LIN {X 0,Y 198.707,Z 605.472,A -85,B 0,C 180,E1 -21893.443,E2 -21893.443} C_VEL
LIN {X 0,Y 202.396,Z 597.043,A -85,B 0,C 180,E1 -21896.831,E2 -21896.831} C_VEL
LIN {X 0,Y 206.089,Z 588.246,A -85,B 0,C 180,E1 -21899.631,E2 -21899.631} C_VEL
LIN {X 0,Y 209.473,Z 579.533,A -85,B 0,C 180,E1 -21901.895,E2 -21901.895} C_VEL
LIN {X 0,Y 213.628,Z 567.883,A -85,B 0,C 180,E1 -21904.308,E2 -21904.308} C_VEL
LIN {X 0,Y 217.053,Z 556.425,A -85,B 0,C 180,E1 -21906.218,E2 -21906.218} C_VEL
LIN {X 0,Y 220.359,Z 543.729,A -85,B 0,C 180,E1 -21907.872,E2 -21907.872} C_VEL
LIN {X 0,Y 223.315,Z 530.569,A -85,B 0,C 180,E1 -21909.149,E2 -21909.149} C_VEL
LIN {X 0,Y 225.4,Z 517.843,A -85,B 0,C 180,E1 -21910.091,E2 -21910.091} C_VEL
LIN {X 0,Y 227.124,Z 503.349,A -85,B 0,C 180,E1 -21910.82,E2 -21910.82} C_VEL
LIN {X 0,Y 231.055,Z 437.728,A -85,B 0,C 180,E1 -21912.715,E2 -21912.715} C_VEL
LIN {X 0,Y 231.07,Z 434.373,A -85,B 0,C 180,E1 -21912.851,E2 -21912.851} C_VEL
LIN {X 0,Y 224.582,Z 419.408,A -85,B 0,C 180,E1 -21915.069,E2 -21915.069} C_VEL
LIN {X 0,Y 218.217,Z 406.943,A -85,B 0,C 180,E1 -21917.363,E2 -21917.363} C_VEL
LIN {X 0,Y 214.281,Z 400.305,A -85,B 0,C 180,E1 -21918.851,E2 -21918.851} C_VEL
LIN {X 0,Y 209.411,Z 393.182,A -85,B 0,C 180,E1 -21920.78,E2 -21920.78} C_VEL
LIN {X 0,Y 206.167,Z 388.687,A -85,B 0,C 180,E1 -21922.149,E2 -21922.149} C_VEL
LIN {X 0,Y 203.479,Z 384.928,A -85,B 0,C 180,E1 -21923.353,E2 -21923.353} C_VEL
LIN {X 0,Y 200.868,Z 381.448,A -85,B 0,C 180,E1 -21924.578,E2 -21924.578} C_VEL
LIN {X 0,Y 199.915,Z 380.302,A -85,B 0,C 180,E1 -21925.035,E2 -21925.035} C_VEL
LIN {X 0,Y 197.517,Z 377.514,A -85,B 0,C 180,E1 -21926.222,E2 -21926.222} C_VEL
LIN {X 0,Y 196.503,Z 375.589,A -85,B 0,C 180,E1 -21926.793,E2 -21926.793} C_VEL
LIN {X 0,Y 194.099,Z 373.615,A -85,B 0,C 180,E1 -21928.031,E2 -21928.031} C_VEL
LIN {X 0,Y 192.852,Z 371.337,A -85,B 0,C 180,E1 -21928.79,E2 -21928.79} C_VEL
LIN {X 0,Y 192.566,Z 370.108,A -85,B 0,C 180,E1 -21929.044,E2 -21929.044} C_VEL
LIN {X 0,Y 192.61,Z 370.098,A -85,B 0,C 180,E1 -21931.683,E2 -21931.683} C_VEL
LIN {X 0,Y 192.662,Z 370.106,A -85,B 0,C 180,E1 -21936.343,E2 -21936.343} C_VEL
LIN {X 0,Y 192.683,Z 370.072,A -85,B 0,C 180,E1 -21941.49,E2 -21941.49} C_VEL
LIN {X 0,Y 192.723,Z 370.103,A -85,B 0,C 180,E1 -21945.21,E2 -21945.21} C_VEL
LIN {X 0,Y 192.933,Z 370.075,A -85,B 0,C 180,E1 -21949.566,E2 -21949.566} C_VEL
LIN {X 0,Y 192.953,Z 370.074,A -85,B 0,C 180,E1 -21953.727,E2 -21953.727} C_VEL
LIN {X 0,Y 193.218,Z 370.043,A -85,B 0,C 180,E1 -21957.915,E2 -21957.915} C_VEL
LIN {X 0,Y 193.4,Z 370.008,A -85,B 0,C 180,E1 -21960,E2 -21960} C_VEL
LIN {X 0,Y 192.923,Z 370.068,A -85,B 0,C 180,E1 -21964.178,E2 -21964.178} C_VEL
LIN {X 0,Y 193.011,Z 370.058,A -85,B 0,C 180,E1 -21968.375,E2 -21968.375} C_VEL
LIN {X 0,Y 192.778,Z 370.087,A -85,B 0,C 180,E1 -21972.635,E2 -21972.635} C_VEL
LIN {X 0,Y 192.704,Z 370.097,A -85,B 0,C 180,E1 -21976.963,E2 -21976.963} C_VEL
LIN {X 0,Y 192.561,Z 370.092,A -85,B 0,C 180,E1 -21981.406,E2 -21981.406} C_VEL
LIN {X 0,Y 192.599,Z 370.097,A -85,B 0,C 180,E1 -21984.19,E2 -21984.19} C_VEL
LIN {X 0,Y 192.589,Z 370.093,A -85,B 0,C 180,E1 -21988.866,E2 -21988.866} C_VEL
LIN {X 0,Y 192.562,Z 370.11,A -85,B 0,C 180,E1 -21990.88,E2 -21990.88} C_VEL
LIN {X 0,Y 193.417,Z 372.657,A -85,B 0,C 180,E1 -21991.489,E2 -21991.489} C_VEL
LIN {X 0,Y 193.705,Z 373.112,A -85,B 0,C 180,E1 -21991.659,E2 -21991.659} C_VEL
LIN {X 0,Y 196.21,Z 378.545,A -85,B 0,C 180,E1 -21993.181,E2 -21993.181} C_VEL
LIN {X 0,Y 202.441,Z 393.008,A -85,B 0,C 180,E1 -21996.634,E2 -21996.634} C_VEL
LIN {X 0,Y 203.994,Z 395.569,A -85,B 0,C 180,E1 -21997.361,E2 -21997.361} C_VEL
LIN {X 0,Y 210.292,Z 406.349,A -85,B 0,C 180,E1 -22000.114,E2 -22000.114} C_VEL
LIN {X 0,Y 216.539,Z 418.079,A -85,B 0,C 180,E1 -22002.6,E2 -22002.6} C_VEL
LIN {X 0,Y 222.539,Z 431.217,A -85,B 0,C 180,E1 -22004.843,E2 -22004.843} C_VEL
LIN {X 0,Y 225.822,Z 439.404,A -85,B 0,C 180,E1 -22006.029,E2 -22006.029} C_VEL
LIN {X 0,Y 221.988,Z 502.379,A -85,B 0,C 180,E1 -22007.846,E2 -22007.846} C_VEL
LIN {X 0,Y 220.45,Z 517.246,A -85,B 0,C 180,E1 -22008.513,E2 -22008.513} C_VEL
LIN {X 0,Y 218.354,Z 529.758,A -85,B 0,C 180,E1 -22009.329,E2 -22009.329} C_VEL
LIN {X 0,Y 215.954,Z 540.985,A -85,B 0,C 180,E1 -22010.311,E2 -22010.311} C_VEL
LIN {X 0,Y 212.766,Z 553.433,A -85,B 0,C 180,E1 -22011.736,E2 -22011.736} C_VEL
LIN {X 0,Y 209.227,Z 565.16,A -85,B 0,C 180,E1 -22013.464,E2 -22013.464} C_VEL
LIN {X 0,Y 205.398,Z 576.632,A -85,B 0,C 180,E1 -22015.632,E2 -22015.632} C_VEL
LIN {X 0,Y 201.599,Z 586.349,A -85,B 0,C 180,E1 -22017.888,E2 -22017.888} C_VEL
LIN {X 0,Y 197.502,Z 596.069,A -85,B 0,C 180,E1 -22020.71,E2 -22020.71} C_VEL
LIN {X 0,Y 193.869,Z 604.134,A -85,B 0,C 180,E1 -22023.639,E2 -22023.639} C_VEL
LIN {X 0,Y 190.425,Z 611.727,A -85,B 0,C 180,E1 -22027.125,E2 -22027.125} C_VEL
LIN {X 0,Y 188.014,Z 617.259,A -85,B 0,C 180,E1 -22030.345,E2 -22030.345} C_VEL
LIN {X 0,Y 185.449,Z 622.939,A -85,B 0,C 180,E1 -22034.62,E2 -22034.62} C_VEL
LIN {X 0,Y 183.947,Z 627.063,A -85,B 0,C 180,E1 -22038.99,E2 -22038.99} C_VEL
LIN {X 0,Y 183.189,Z 629.751,A -85,B 0,C 180,E1 -22043.394,E2 -22043.394} C_VEL
LIN {X 0,Y 182.991,Z 631.077,A -85,B 0,C 180,E1 -22047.802,E2 -22047.802} C_VEL
LIN {X 0,Y 183.062,Z 631.239,A -85,B 0,C 180,E1 -22050.003,E2 -22050.003} C_VEL
LIN {X 0,Y 183.019,Z 630.557,A -85,B 0,C 180,E1 -22054.408,E2 -22054.408} C_VEL
LIN {X 0,Y 183.498,Z 628.531,A -85,B 0,C 180,E1 -22058.816,E2 -22058.816} C_VEL
LIN {X 0,Y 184.614,Z 625.117,A -85,B 0,C 180,E1 -22063.207,E2 -22063.207} C_VEL
LIN {X 0,Y 186.675,Z 620.215,A -85,B 0,C 180,E1 -22067.532,E2 -22067.532} C_VEL
LIN {X 0,Y 189.593,Z 613.67,A -85,B 0,C 180,E1 -22071.761,E2 -22071.761} C_VEL
LIN {X 0,Y 193.917,Z 611.789,A -85,B 0,C 180,E1 -22075.783,E2 -22075.783} C_VEL
LIN {X 0,Y 199.616,Z 608.772,A -85,B 0,C 180,E1 -22079.535,E2 -22079.535} C_VEL
LIN {X 0,Y 206.41,Z 604.439,A -85,B 0,C 180,E1 -22083.013,E2 -22083.013} C_VEL
LIN {X 0,Y 214.305,Z 598.674,A -85,B 0,C 180,E1 -22086.181,E2 -22086.181} C_VEL
LIN {X 0,Y 223.09,Z 591.287,A -85,B 0,C 180,E1 -22089.058,E2 -22089.058} C_VEL
LIN {X 0,Y 232.751,Z 582.111,A -85,B 0,C 180,E1 -22091.631,E2 -22091.631} C_VEL
LIN {X 0,Y 241.882,Z 572.221,A -85,B 0,C 180,E1 -22093.638,E2 -22093.638} C_VEL
LIN {X 0,Y 250.221,Z 562.013,A -85,B 0,C 180,E1 -22095.165,E2 -22095.165} C_VEL
LIN {X 0,Y 257.281,Z 552.141,A -85,B 0,C 180,E1 -22096.279,E2 -22096.279} C_VEL
LIN {X 0,Y 257.573,Z 551.734,A -85,B 0,C 180,E1 -22096.657,E2 -22096.657} C_VEL
LIN {X 0,Y 250.018,Z 562.221,A -85,B 0,C 180,E1 -22098.117,E2 -22098.117} C_VEL
LIN {X 0,Y 242.233,Z 571.531,A -85,B 0,C 180,E1 -22099.793,E2 -22099.793} C_VEL
LIN {X 0,Y 233.601,Z 580.397,A -85,B 0,C 180,E1 -22101.921,E2 -22101.921} C_VEL
LIN {X 0,Y 225.099,Z 587.859,A -85,B 0,C 180,E1 -22104.335,E2 -22104.335} C_VEL
LIN {X 0,Y 217.934,Z 593.201,A -85,B 0,C 180,E1 -22106.755,E2 -22106.755} C_VEL
LIN {X 0,Y 210.044,Z 598.033,A -85,B 0,C 180,E1 -22109.875,E2 -22109.875} C_VEL
LIN {X 0,Y 203.096,Z 601.298,A -85,B 0,C 180,E1 -22113.266,E2 -22113.266} C_VEL
LIN {X 0,Y 197.064,Z 603.056,A -85,B 0,C 180,E1 -22116.903,E2 -22116.903} C_VEL
LIN {X 0,Y 192.029,Z 603.407,A -85,B 0,C 180,E1 -22120.769,E2 -22120.769} C_VEL
LIN {X 0,Y 188.438,Z 602.296,A -85,B 0,C 180,E1 -22124.866,E2 -22124.866} C_VEL
LIN {X 0,Y 185.775,Z 599.724,A -85,B 0,C 180,E1 -22129.097,E2 -22129.097} C_VEL
LIN {X 0,Y 184.203,Z 595.669,A -85,B 0,C 180,E1 -22133.428,E2 -22133.428} C_VEL
LIN {X 0,Y 183.814,Z 591.518,A -85,B 0,C 180,E1 -22136.712,E2 -22136.712} C_VEL
LIN {X 0,Y 183.676,Z 585.283,A -85,B 0,C 180,E1 -22140.548,E2 -22140.548} C_VEL
LIN {X 0,Y 183.852,Z 578.541,A -85,B 0,C 180,E1 -22143.836,E2 -22143.836} C_VEL
LIN {X 0,Y 184.278,Z 570.082,A -85,B 0,C 180,E1 -22147.175,E2 -22147.175} C_VEL
LIN {X 0,Y 184.92,Z 559.88,A -85,B 0,C 180,E1 -22150.401,E2 -22150.401} C_VEL
LIN {X 0,Y 185.69,Z 549.274,A -85,B 0,C 180,E1 -22153.126,E2 -22153.126} C_VEL
LIN {X 0,Y 186.702,Z 537.558,A -85,B 0,C 180,E1 -22155.558,E2 -22155.558} C_VEL
LIN {X 0,Y 187.729,Z 524.558,A -85,B 0,C 180,E1 -22157.709,E2 -22157.709} C_VEL
LIN {X 0,Y 188.701,Z 510.981,A -85,B 0,C 180,E1 -22159.443,E2 -22159.443} C_VEL
LIN {X 0,Y 189.583,Z 495.968,A -85,B 0,C 180,E1 -22160.833,E2 -22160.833} C_VEL
LIN {X 0,Y 193.383,Z 417.044,A -85,B 0,C 180,E1 -22166.116,E2 -22166.116} C_VEL
LIN {X 0,Y 191.04,Z 396.091,A -85,B 0,C 180,E1 -22167.576,E2 -22167.576} C_VEL
LIN {X 0,Y 188.706,Z 385.709,A -85,B 0,C 180,E1 -22168.414,E2 -22168.414} C_VEL
LIN {X 0,Y 187.873,Z 381.706,A -85,B 0,C 180,E1 -22169.657,E2 -22169.657} C_VEL
LIN {X 0,Y 188.604,Z 383.232,A -85,B 0,C 180,E1 -22170.16,E2 -22170.16} C_VEL
LIN {X 0,Y 189.272,Z 383.585,A -85,B 0,C 180,E1 -22170.533,E2 -22170.533} C_VEL
LIN {X 0,Y 191.035,Z 383.228,A -85,B 0,C 180,E1 -22171.395,E2 -22171.395} C_VEL
LIN {X 0,Y 192.098,Z 382.434,A -85,B 0,C 180,E1 -22171.858,E2 -22171.858} C_VEL
LIN {X 0,Y 194.344,Z 382.672,A -85,B 0,C 180,E1 -22172.927,E2 -22172.927} C_VEL
LIN {X 0,Y 197.017,Z 386.201,A -85,B 0,C 180,E1 -22174.338,E2 -22174.338} C_VEL
LIN {X 0,Y 198.275,Z 387.839,A -85,B 0,C 180,E1 -22174.97,E2 -22174.97} C_VEL
LIN {X 0,Y 201.836,Z 392.677,A -85,B 0,C 180,E1 -22176.678,E2 -22176.678} C_VEL
LIN {X 0,Y 207.332,Z 400.427,A -85,B 0,C 180,E1 -22179.097,E2 -22179.097} C_VEL
LIN {X 0,Y 212.843,Z 409.078,A -85,B 0,C 180,E1 -22181.33,E2 -22181.33} C_VEL
LIN {X 0,Y 219.414,Z 422.009,A -85,B 0,C 180,E1 -22183.854,E2 -22183.854} C_VEL
LIN {X 0,Y 224.284,Z 433.17,A -85,B 0,C 180,E1 -22185.63,E2 -22185.63} C_VEL
LIN {X 0,Y 225.739,Z 436.684,A -85,B 0,C 180,E1 -22186.144,E2 -22186.144} C_VEL
LIN {X 0,Y 223.107,Z 481.871,A -85,B 0,C 180,E1 -22187.457,E2 -22187.457} C_VEL
LIN {X 0,Y 221.59,Z 504.39,A -85,B 0,C 180,E1 -22188.162,E2 -22188.162} C_VEL
LIN {X 0,Y 219.962,Z 517.73,A -85,B 0,C 180,E1 -22188.85,E2 -22188.85} C_VEL
LIN {X 0,Y 217.444,Z 531.634,A -85,B 0,C 180,E1 -22189.876,E2 -22189.876} C_VEL
LIN {X 0,Y 214.505,Z 544.565,A -85,B 0,C 180,E1 -22191.197,E2 -22191.197} C_VEL
LIN {X 0,Y 211.033,Z 557.109,A -85,B 0,C 180,E1 -22192.868,E2 -22192.868} C_VEL
LIN {X 0,Y 207.451,Z 568.548,A -85,B 0,C 180,E1 -22194.833,E2 -22194.833} C_VEL
LIN {X 0,Y 203.572,Z 579.047,A -85,B 0,C 180,E1 -22197.058,E2 -22197.058} C_VEL
LIN {X 0,Y 200.001,Z 587.851,A -85,B 0,C 180,E1 -22199.365,E2 -22199.365} C_VEL
LIN {X 0,Y 196.155,Z 596.725,A -85,B 0,C 180,E1 -22202.237,E2 -22202.237} C_VEL
LIN {X 0,Y 192.286,Z 605.219,A -85,B 0,C 180,E1 -22205.718,E2 -22205.718} C_VEL
LIN {X 0,Y 189.301,Z 612.061,A -85,B 0,C 180,E1 -22209.344,E2 -22209.344} C_VEL
LIN {X 0,Y 187.046,Z 616.782,A -85,B 0,C 180,E1 -22212.504,E2 -22212.504} C_VEL
LIN {X 0,Y 184.936,Z 621.666,A -85,B 0,C 180,E1 -22216.817,E2 -22216.817} C_VEL
LIN {X 0,Y 183.702,Z 625.064,A -85,B 0,C 180,E1 -22221.194,E2 -22221.194} C_VEL
LIN {X 0,Y 183.125,Z 627.082,A -85,B 0,C 180,E1 -22225.595,E2 -22225.595} C_VEL
LIN {X 0,Y 183.07,Z 627.769,A -85,B 0,C 180,E1 -22229.997,E2 -22229.997} C_VEL
LIN {X 0,Y 183.123,Z 627.138,A -85,B 0,C 180,E1 -22234.399,E2 -22234.399} C_VEL
LIN {X 0,Y 183.681,Z 625.172,A -85,B 0,C 180,E1 -22238.8,E2 -22238.8} C_VEL
LIN {X 0,Y 184.896,Z 621.821,A -85,B 0,C 180,E1 -22243.18,E2 -22243.18} C_VEL
LIN {X 0,Y 187.015,Z 616.983,A -85,B 0,C 180,E1 -22247.492,E2 -22247.492} C_VEL
LIN {X 0,Y 189.191,Z 612.318,A -85,B 0,C 180,E1 -22250.661,E2 -22250.661} C_VEL
LIN {X 0,Y 192.191,Z 605.537,A -85,B 0,C 180,E1 -22254.288,E2 -22254.288} C_VEL
LIN {X 0,Y 196.076,Z 597.108,A -85,B 0,C 180,E1 -22257.769,E2 -22257.769} C_VEL
LIN {X 0,Y 199.924,Z 588.311,A -85,B 0,C 180,E1 -22260.641,E2 -22260.641} C_VEL
LIN {X 0,Y 203.474,Z 579.598,A -85,B 0,C 180,E1 -22262.953,E2 -22262.953} C_VEL
LIN {X 0,Y 207.381,Z 569.207,A -85,B 0,C 180,E1 -22265.174,E2 -22265.174} C_VEL
LIN {X 0,Y 210.943,Z 557.912,A -85,B 0,C 180,E1 -22267.143,E2 -22267.143} C_VEL
LIN {X 0,Y 214.35,Z 545.556,A -85,B 0,C 180,E1 -22268.829,E2 -22268.829} C_VEL
LIN {X 0,Y 217.371,Z 532.887,A -85,B 0,C 180,E1 -22270.133,E2 -22270.133} C_VEL
LIN {X 0,Y 219.793,Z 519.423,A -85,B 0,C 180,E1 -22271.181,E2 -22271.181} C_VEL
LIN {X 0,Y 221.572,Z 505.563,A -85,B 0,C 180,E1 -22271.927,E2 -22271.927} C_VEL
LIN {X 0,Y 223.066,Z 485.36,A -85,B 0,C 180,E1 -22272.567,E2 -22272.567} C_VEL
LIN {X 0,Y 225.873,Z 436.775,A -85,B 0,C 180,E1 -22273.984,E2 -22273.984} C_VEL
LIN {X 0,Y 219.558,Z 422.15,A -85,B 0,C 180,E1 -22276.274,E2 -22276.274} C_VEL
LIN {X 0,Y 212.497,Z 408.401,A -85,B 0,C 180,E1 -22278.995,E2 -22278.995} C_VEL
LIN {X 0,Y 206.716,Z 399.463,A -85,B 0,C 180,E1 -22281.362,E2 -22281.362} C_VEL
LIN {X 0,Y 200.489,Z 390.766,A -85,B 0,C 180,E1 -22284.168,E2 -22284.168} C_VEL
LIN {X 0,Y 197.112,Z 386.299,A -85,B 0,C 180,E1 -22285.836,E2 -22285.836} C_VEL
LIN {X 0,Y 194.47,Z 382.927,A -85,B 0,C 180,E1 -22287.227,E2 -22287.227} C_VEL
LIN {X 0,Y 193.636,Z 381.69,A -85,B 0,C 180,E1 -22287.697,E2 -22287.697} C_VEL
LIN {X 0,Y 191.036,Z 378.928,A -85,B 0,C 180,E1 -22289.153,E2 -22289.153} C_VEL
LIN {X 0,Y 189.725,Z 376.624,A -85,B 0,C 180,E1 -22289.994,E2 -22289.994} C_VEL
LIN {X 0,Y 187.341,Z 374.834,A -85,B 0,C 180,E1 -22291.425,E2 -22291.425} C_VEL
LIN {X 0,Y 185.853,Z 372.39,A -85,B 0,C 180,E1 -22292.48,E2 -22292.48} C_VEL
LIN {X 0,Y 185.509,Z 370.971,A -85,B 0,C 180,E1 -22292.883,E2 -22292.883} C_VEL
LIN {X 0,Y 185.57,Z 370.973,A -85,B 0,C 180,E1 -22295.38,E2 -22295.38} C_VEL
LIN {X 0,Y 185.614,Z 370.95,A -85,B 0,C 180,E1 -22301.177,E2 -22301.177} C_VEL
LIN {X 0,Y 185.652,Z 370.986,A -85,B 0,C 180,E1 -22304.633,E2 -22304.633} C_VEL
LIN {X 0,Y 185.876,Z 370.955,A -85,B 0,C 180,E1 -22309.418,E2 -22309.418} C_VEL
LIN {X 0,Y 185.918,Z 370.952,A -85,B 0,C 180,E1 -22313.488,E2 -22313.488} C_VEL
LIN {X 0,Y 186.164,Z 370.922,A -85,B 0,C 180,E1 -22317.836,E2 -22317.836} C_VEL
LIN {X 0,Y 186.366,Z 370.884,A -85,B 0,C 180,E1 -22320,E2 -22320} C_VEL
LIN {X 0,Y 185.871,Z 370.946,A -85,B 0,C 180,E1 -22324.337,E2 -22324.337} C_VEL
LIN {X 0,Y 185.961,Z 370.936,A -85,B 0,C 180,E1 -22328.695,E2 -22328.695} C_VEL
LIN {X 0,Y 185.704,Z 370.968,A -85,B 0,C 180,E1 -22333.125,E2 -22333.125} C_VEL
LIN {X 0,Y 185.641,Z 370.978,A -85,B 0,C 180,E1 -22337.63,E2 -22337.63} C_VEL
LIN {X 0,Y 185.528,Z 370.965,A -85,B 0,C 180,E1 -22342.26,E2 -22342.26} C_VEL
LIN {X 0,Y 185.513,Z 371.02,A -85,B 0,C 180,E1 -22347.116,E2 -22347.116} C_VEL
LIN {X 0,Y 186.269,Z 373.389,A -85,B 0,C 180,E1 -22347.758,E2 -22347.758} C_VEL
LIN {X 0,Y 188.414,Z 375.851,A -85,B 0,C 180,E1 -22349.159,E2 -22349.159} C_VEL
LIN {X 0,Y 189.937,Z 376.846,A -85,B 0,C 180,E1 -22350.045,E2 -22350.045} C_VEL
LIN {X 0,Y 191.839,Z 380.019,A -85,B 0,C 180,E1 -22351.236,E2 -22351.236} C_VEL
LIN {X 0,Y 194.171,Z 382.365,A -85,B 0,C 180,E1 -22352.509,E2 -22352.509} C_VEL
LIN {X 0,Y 196.68,Z 385.884,A -85,B 0,C 180,E1 -22353.863,E2 -22353.863} C_VEL
LIN {X 0,Y 198.116,Z 387.577,A -85,B 0,C 180,E1 -22354.582,E2 -22354.582} C_VEL
LIN {X 0,Y 201.825,Z 392.601,A -85,B 0,C 180,E1 -22356.375,E2 -22356.375} C_VEL
LIN {X 0,Y 203.994,Z 395.569,A -85,B 0,C 180,E1 -22357.361,E2 -22357.361} C_VEL
LIN {X 0,Y 206.102,Z 399.752,A -85,B 0,C 180,E1 -22358.352,E2 -22358.352} C_VEL
LIN {X 0,Y 207.66,Z 404.671,A -85,B 0,C 180,E1 -22359.155,E2 -22359.155} C_VEL
LIN {X 0,Y 211.072,Z 418.814,A -85,B 0,C 180,E1 -22361.001,E2 -22361.001} C_VEL
LIN {X 0,Y 212.243,Z 422.12,A -85,B 0,C 180,E1 -22361.528,E2 -22361.528} C_VEL
LIN {X 0,Y 217.855,Z 434.676,A -85,B 0,C 180,E1 -22363.755,E2 -22363.755} C_VEL
LIN {X 0,Y 220.59,Z 441.582,A -85,B 0,C 180,E1 -22364.803,E2 -22364.803} C_VEL
LIN {X 0,Y 217.065,Z 498.535,A -85,B 0,C 180,E1 -22366.462,E2 -22366.462} C_VEL
LIN {X 0,Y 215.781,Z 512.612,A -85,B 0,C 180,E1 -22367.009,E2 -22367.009} C_VEL
LIN {X 0,Y 213.471,Z 527.097,A -85,B 0,C 180,E1 -22367.876,E2 -22367.876} C_VEL
LIN {X 0,Y 210.538,Z 540.924,A -85,B 0,C 180,E1 -22369.077,E2 -22369.077} C_VEL
LIN {X 0,Y 207.238,Z 553.371,A -85,B 0,C 180,E1 -22370.52,E2 -22370.52} C_VEL
LIN {X 0,Y 203.199,Z 566.134,A -85,B 0,C 180,E1 -22372.445,E2 -22372.445} C_VEL
LIN {X 0,Y 199.14,Z 577.725,A -85,B 0,C 180,E1 -22374.726,E2 -22374.726} C_VEL
LIN {X 0,Y 194.825,Z 588.067,A -85,B 0,C 180,E1 -22377.245,E2 -22377.245} C_VEL
LIN {X 0,Y 190.651,Z 597.489,A -85,B 0,C 180,E1 -22380.159,E2 -22380.159} C_VEL
LIN {X 0,Y 186.357,Z 606.463,A -85,B 0,C 180,E1 -22383.701,E2 -22383.701} C_VEL
LIN {X 0,Y 182.895,Z 613.717,A -85,B 0,C 180,E1 -22387.406,E2 -22387.406} C_VEL
LIN {X 0,Y 180.578,Z 618.802,A -85,B 0,C 180,E1 -22390.686,E2 -22390.686} C_VEL
LIN {X 0,Y 178.065,Z 624.051,A -85,B 0,C 180,E1 -22395.138,E2 -22395.138} C_VEL
LIN {X 0,Y 176.951,Z 626.996,A -85,B 0,C 180,E1 -22398.549,E2 -22398.549} C_VEL
LIN {X 0,Y 176.121,Z 629.684,A -85,B 0,C 180,E1 -22403.128,E2 -22403.128} C_VEL
LIN {X 0,Y 175.886,Z 631.01,A -85,B 0,C 180,E1 -22407.713,E2 -22407.713} C_VEL
LIN {X 0,Y 175.974,Z 631.172,A -85,B 0,C 180,E1 -22410.003,E2 -22410.003} C_VEL
LIN {X 0,Y 175.942,Z 630.489,A -85,B 0,C 180,E1 -22414.586,E2 -22414.586} C_VEL
LIN {X 0,Y 176.456,Z 628.463,A -85,B 0,C 180,E1 -22419.17,E2 -22419.17} C_VEL
LIN {X 0,Y 177.669,Z 625.049,A -85,B 0,C 180,E1 -22423.733,E2 -22423.733} C_VEL
LIN {X 0,Y 179.889,Z 620.147,A -85,B 0,C 180,E1 -22428.216,E2 -22428.216} C_VEL
LIN {X 0,Y 182.95,Z 613.6,A -85,B 0,C 180,E1 -22432.594,E2 -22432.594} C_VEL
LIN {X 0,Y 183.345,Z 613.131,A -85,B 0,C 180,E1 -22433.078,E2 -22433.078} C_VEL
LIN {X 0,Y 187.556,Z 611.935,A -85,B 0,C 180,E1 -22436.725,E2 -22436.725} C_VEL
LIN {X 0,Y 193.492,Z 609.399,A -85,B 0,C 180,E1 -22440.568,E2 -22440.568} C_VEL
LIN {X 0,Y 200.573,Z 605.603,A -85,B 0,C 180,E1 -22444.103,E2 -22444.103} C_VEL
LIN {X 0,Y 208.767,Z 600.448,A -85,B 0,C 180,E1 -22447.301,E2 -22447.301} C_VEL
LIN {X 0,Y 217.872,Z 593.752,A -85,B 0,C 180,E1 -22450.18,E2 -22450.18} C_VEL
LIN {X 0,Y 227.814,Z 585.408,A -85,B 0,C 180,E1 -22452.745,E2 -22452.745} C_VEL
LIN {X 0,Y 236.067,Z 577.561,A -85,B 0,C 180,E1 -22454.519,E2 -22454.519} C_VEL
LIN {X 0,Y 245.567,Z 567.308,A -85,B 0,C 180,E1 -22456.232,E2 -22456.232} C_VEL
LIN {X 0,Y 246.939,Z 565.744,A -85,B 0,C 180,E1 -22456.447,E2 -22456.447} C_VEL
LIN {X 0,Y 246.766,Z 565.945,A -85,B 0,C 180,E1 -22456.88,E2 -22456.88} C_VEL
LIN {X 0,Y 237.376,Z 575.964,A -85,B 0,C 180,E1 -22458.795,E2 -22458.795} C_VEL
LIN {X 0,Y 228.45,Z 584.03,A -85,B 0,C 180,E1 -22460.901,E2 -22460.901} C_VEL
LIN {X 0,Y 219.702,Z 590.763,A -85,B 0,C 180,E1 -22463.318,E2 -22463.318} C_VEL
LIN {X 0,Y 212.302,Z 595.566,A -85,B 0,C 180,E1 -22465.753,E2 -22465.753} C_VEL
LIN {X 0,Y 204.104,Z 599.804,A -85,B 0,C 180,E1 -22468.902,E2 -22468.902} C_VEL
LIN {X 0,Y 196.881,Z 602.546,A -85,B 0,C 180,E1 -22472.351,E2 -22472.351} C_VEL
LIN {X 0,Y 190.595,Z 603.849,A -85,B 0,C 180,E1 -22476.07,E2 -22476.07} C_VEL
LIN {X 0,Y 185.351,Z 603.725,A -85,B 0,C 180,E1 -22480.047,E2 -22480.047} C_VEL
LIN {X 0,Y 181.613,Z 602.206,A -85,B 0,C 180,E1 -22484.283,E2 -22484.283} C_VEL
LIN {X 0,Y 178.844,Z 599.248,A -85,B 0,C 180,E1 -22488.669,E2 -22488.669} C_VEL
LIN {X 0,Y 177.224,Z 594.76,A -85,B 0,C 180,E1 -22493.168,E2 -22493.168} C_VEL
LIN {X 0,Y 176.834,Z 590.321,A -85,B 0,C 180,E1 -22496.582,E2 -22496.582} C_VEL
LIN {X 0,Y 176.706,Z 583.717,A -85,B 0,C 180,E1 -22500.57,E2 -22500.57} C_VEL
LIN {X 0,Y 176.888,Z 576.582,A -85,B 0,C 180,E1 -22503.987,E2 -22503.987} C_VEL
LIN {X 0,Y 177.34,Z 567.678,A -85,B 0,C 180,E1 -22507.43,E2 -22507.43} C_VEL
LIN {X 0,Y 177.931,Z 558.851,A -85,B 0,C 180,E1 -22510.239,E2 -22510.239} C_VEL
LIN {X 0,Y 178.726,Z 547.953,A -85,B 0,C 180,E1 -22513.068,E2 -22513.068} C_VEL
LIN {X 0,Y 179.734,Z 536.008,A -85,B 0,C 180,E1 -22515.595,E2 -22515.595} C_VEL
LIN {X 0,Y 180.8,Z 522.531,A -85,B 0,C 180,E1 -22517.825,E2 -22517.825} C_VEL
LIN {X 0,Y 181.786,Z 508.23,A -85,B 0,C 180,E1 -22519.625,E2 -22519.625} C_VEL
LIN {X 0,Y 182.545,Z 494.845,A -85,B 0,C 180,E1 -22520.863,E2 -22520.863} C_VEL
LIN {X 0,Y 186.308,Z 417.588,A -85,B 0,C 180,E1 -22526.292,E2 -22526.292} C_VEL
LIN {X 0,Y 184.132,Z 397.564,A -85,B 0,C 180,E1 -22527.74,E2 -22527.74} C_VEL
LIN {X 0,Y 183.291,Z 393.818,A -85,B 0,C 180,E1 -22528.033,E2 -22528.033} C_VEL
LIN {X 0,Y 183.836,Z 394.891,A -85,B 0,C 180,E1 -22528.438,E2 -22528.438} C_VEL
LIN {X 0,Y 185.317,Z 394.673,A -85,B 0,C 180,E1 -22529.258,E2 -22529.258} C_VEL
LIN {X 0,Y 186.79,Z 392.34,A -85,B 0,C 180,E1 -22529.882,E2 -22529.882} C_VEL
LIN {X 0,Y 187.698,Z 390.454,A -85,B 0,C 180,E1 -22530.222,E2 -22530.222} C_VEL
LIN {X 0,Y 190.479,Z 390.401,A -85,B 0,C 180,E1 -22531.63,E2 -22531.63} C_VEL
LIN {X 0,Y 192.248,Z 389.61,A -85,B 0,C 180,E1 -22532.424,E2 -22532.424} C_VEL
LIN {X 0,Y 195.629,Z 394.039,A -85,B 0,C 180,E1 -22534.241,E2 -22534.241} C_VEL
LIN {X 0,Y 199.148,Z 398.873,A -85,B 0,C 180,E1 -22535.999,E2 -22535.999} C_VEL
LIN {X 0,Y 206.019,Z 408.894,A -85,B 0,C 180,E1 -22539.106,E2 -22539.106} C_VEL
LIN {X 0,Y 210.05,Z 415.918,A -85,B 0,C 180,E1 -22540.806,E2 -22540.806} C_VEL
LIN {X 0,Y 216.135,Z 428.322,A -85,B 0,C 180,E1 -22543.24,E2 -22543.24} C_VEL
LIN {X 0,Y 220.586,Z 439.117,A -85,B 0,C 180,E1 -22544.949,E2 -22544.949} C_VEL
LIN {X 0,Y 216.585,Z 502.522,A -85,B 0,C 180,E1 -22546.832,E2 -22546.832} C_VEL
LIN {X 0,Y 214.902,Z 516.282,A -85,B 0,C 180,E1 -22547.502,E2 -22547.502} C_VEL
LIN {X 0,Y 212.298,Z 530.58,A -85,B 0,C 180,E1 -22548.537,E2 -22548.537} C_VEL
LIN {X 0,Y 209.478,Z 542.875,A -85,B 0,C 180,E1 -22549.768,E2 -22549.768} C_VEL
LIN {X 0,Y 205.826,Z 555.757,A -85,B 0,C 180,E1 -22551.45,E2 -22551.45} C_VEL
LIN {X 0,Y 202.387,Z 566.646,A -85,B 0,C 180,E1 -22553.296,E2 -22553.296} C_VEL
LIN {X 0,Y 198.44,Z 577.17,A -85,B 0,C 180,E1 -22555.479,E2 -22555.479} C_VEL
LIN {X 0,Y 194.579,Z 586.298,A -85,B 0,C 180,E1 -22557.805,E2 -22557.805} C_VEL
LIN {X 0,Y 190.539,Z 595.443,A -85,B 0,C 180,E1 -22560.74,E2 -22560.74} C_VEL
LIN {X 0,Y 186.885,Z 603.062,A -85,B 0,C 180,E1 -22563.773,E2 -22563.773} C_VEL
LIN {X 0,Y 183.481,Z 610.326,A -85,B 0,C 180,E1 -22567.475,E2 -22567.475} C_VEL
LIN {X 0,Y 181.021,Z 615.412,A -85,B 0,C 180,E1 -22570.728,E2 -22570.728} C_VEL
LIN {X 0,Y 178.958,Z 619.488,A -85,B 0,C 180,E1 -22574.041,E2 -22574.041} C_VEL
LIN {X 0,Y 177.234,Z 623.611,A -85,B 0,C 180,E1 -22578.561,E2 -22578.561} C_VEL
LIN {X 0,Y 176.319,Z 626.308,A -85,B 0,C 180,E1 -22583.129,E2 -22583.129} C_VEL
LIN {X 0,Y 175.95,Z 627.658,A -85,B 0,C 180,E1 -22587.707,E2 -22587.707} C_VEL
LIN {X 0,Y 175.983,Z 627.836,A -85,B 0,C 180,E1 -22589.997,E2 -22589.997} C_VEL
LIN {X 0,Y 176.034,Z 627.205,A -85,B 0,C 180,E1 -22594.576,E2 -22594.576} C_VEL
LIN {X 0,Y 176.313,Z 626.391,A -85,B 0,C 180,E1 -22596.864,E2 -22596.864} C_VEL
LIN {X 0,Y 177.205,Z 623.742,A -85,B 0,C 180,E1 -22601.434,E2 -22601.434} C_VEL
LIN {X 0,Y 178.927,Z 619.663,A -85,B 0,C 180,E1 -22605.955,E2 -22605.955} C_VEL
LIN {X 0,Y 181.755,Z 614.03,A -85,B 0,C 180,E1 -22610.362,E2 -22610.362} C_VEL
LIN {X 0,Y 184.417,Z 608.237,A -85,B 0,C 180,E1 -22613.847,E2 -22613.847} C_VEL
LIN {X 0,Y 187.949,Z 600.999,A -85,B 0,C 180,E1 -22617.258,E2 -22617.258} C_VEL
LIN {X 0,Y 191.751,Z 592.98,A -85,B 0,C 180,E1 -22620.258,E2 -22620.258} C_VEL
LIN {X 0,Y 196.031,Z 583.309,A -85,B 0,C 180,E1 -22623.139,E2 -22623.139} C_VEL
LIN {X 0,Y 200.381,Z 572.573,A -85,B 0,C 180,E1 -22625.664,E2 -22625.664} C_VEL
LIN {X 0,Y 204.13,Z 561.583,A -85,B 0,C 180,E1 -22627.759,E2 -22627.759} C_VEL
LIN {X 0,Y 207.98,Z 548.982,A -85,B 0,C 180,E1 -22629.625,E2 -22629.625} C_VEL
LIN {X 0,Y 211.223,Z 536.203,A -85,B 0,C 180,E1 -22631.078,E2 -22631.078} C_VEL
LIN {X 0,Y 213.886,Z 523.163,A -85,B 0,C 180,E1 -22632.182,E2 -22632.182} C_VEL
LIN {X 0,Y 215.997,Z 509.188,A -85,B 0,C 180,E1 -22633.017,E2 -22633.017} C_VEL
LIN {X 0,Y 217.292,Z 494.603,A -85,B 0,C 180,E1 -22633.569,E2 -22633.569} C_VEL
LIN {X 0,Y 220.743,Z 439.206,A -85,B 0,C 180,E1 -22635.176,E2 -22635.176} C_VEL
LIN {X 0,Y 215.121,Z 426.013,A -85,B 0,C 180,E1 -22637.339,E2 -22637.339} C_VEL
LIN {X 0,Y 208.292,Z 412.541,A -85,B 0,C 180,E1 -22640.127,E2 -22640.127} C_VEL
LIN {X 0,Y 202.438,Z 403.623,A -85,B 0,C 180,E1 -22642.666,E2 -22642.666} C_VEL
LIN {X 0,Y 197.613,Z 396.622,A -85,B 0,C 180,E1 -22644.976,E2 -22644.976} C_VEL
LIN {X 0,Y 194.099,Z 391.975,A -85,B 0,C 180,E1 -22646.794,E2 -22646.794} C_VEL
LIN {X 0,Y 190.99,Z 387.773,A -85,B 0,C 180,E1 -22648.545,E2 -22648.545} C_VEL
LIN {X 0,Y 188.326,Z 384.629,A -85,B 0,C 180,E1 -22650.134,E2 -22650.134} C_VEL
LIN {X 0,Y 187.308,Z 383.023,A -85,B 0,C 180,E1 -22650.805,E2 -22650.805} C_VEL
LIN {X 0,Y 184.696,Z 380.581,A -85,B 0,C 180,E1 -22652.494,E2 -22652.494} C_VEL
LIN {X 0,Y 183,Z 377.623,A -85,B 0,C 180,E1 -22653.791,E2 -22653.791} C_VEL
LIN {X 0,Y 180.368,Z 375.832,A -85,B 0,C 180,E1 -22655.717,E2 -22655.717} C_VEL
LIN {X 0,Y 178.893,Z 373.53,A -85,B 0,C 180,E1 -22657.02,E2 -22657.02} C_VEL
LIN {X 0,Y 178.513,Z 371.869,A -85,B 0,C 180,E1 -22657.58,E2 -22657.58} C_VEL
LIN {X 0,Y 178.595,Z 371.826,A -85,B 0,C 180,E1 -22661.65,E2 -22661.65} C_VEL
LIN {X 0,Y 178.63,Z 371.85,A -85,B 0,C 180,E1 -22666.345,E2 -22666.345} C_VEL
LIN {X 0,Y 178.892,Z 371.816,A -85,B 0,C 180,E1 -22670.959,E2 -22670.959} C_VEL
LIN {X 0,Y 179.112,Z 371.8,A -85,B 0,C 180,E1 -22677.751,E2 -22677.751} C_VEL
LIN {X 0,Y 179.331,Z 371.76,A -85,B 0,C 180,E1 -22680,E2 -22680} C_VEL
LIN {X 0,Y 178.82,Z 371.825,A -85,B 0,C 180,E1 -22684.508,E2 -22684.508} C_VEL
LIN {X 0,Y 178.892,Z 371.816,A -85,B 0,C 180,E1 -22689.041,E2 -22689.041} C_VEL
LIN {X 0,Y 178.63,Z 371.851,A -85,B 0,C 180,E1 -22693.654,E2 -22693.654} C_VEL
LIN {X 0,Y 178.543,Z 371.867,A -85,B 0,C 180,E1 -22699.153,E2 -22699.153} C_VEL
LIN {X 0,Y 178.499,Z 371.878,A -85,B 0,C 180,E1 -22702.422,E2 -22702.422} C_VEL
LIN {X 0,Y 179.106,Z 374.04,A -85,B 0,C 180,E1 -22703.103,E2 -22703.103} C_VEL
LIN {X 0,Y 180.766,Z 376.25,A -85,B 0,C 180,E1 -22704.513,E2 -22704.513} C_VEL
LIN {X 0,Y 183.185,Z 377.832,A -85,B 0,C 180,E1 -22706.257,E2 -22706.257} C_VEL
LIN {X 0,Y 184.876,Z 380.806,A -85,B 0,C 180,E1 -22707.543,E2 -22707.543} C_VEL
LIN {X 0,Y 187.697,Z 383.55,A -85,B 0,C 180,E1 -22709.359,E2 -22709.359} C_VEL
LIN {X 0,Y 190.198,Z 387.037,A -85,B 0,C 180,E1 -22710.921,E2 -22710.921} C_VEL
LIN {X 0,Y 191.732,Z 388.757,A -85,B 0,C 180,E1 -22711.796,E2 -22711.796} C_VEL
LIN {X 0,Y 194.438,Z 392.348,A -85,B 0,C 180,E1 -22713.295,E2 -22713.295} C_VEL
LIN {X 0,Y 199.028,Z 398.659,A -85,B 0,C 180,E1 -22715.638,E2 -22715.638} C_VEL
LIN {X 0,Y 201.514,Z 402.409,A -85,B 0,C 180,E1 -22716.829,E2 -22716.829} C_VEL
LIN {X 0,Y 206.842,Z 411.774,A -85,B 0,C 180,E1 -22719.259,E2 -22719.259} C_VEL
LIN {X 0,Y 212.243,Z 422.12,A -85,B 0,C 180,E1 -22721.528,E2 -22721.528} C_VEL
LIN {X 0,Y 213.19,Z 425.573,A -85,B 0,C 180,E1 -22721.984,E2 -22721.984} C_VEL
LIN {X 0,Y 213.736,Z 431.992,A -85,B 0,C 180,E1 -22722.46,E2 -22722.46} C_VEL
LIN {X 0,Y 214.319,Z 439.809,A -85,B 0,C 180,E1 -22723.007,E2 -22723.007} C_VEL
LIN {X 0,Y 214.883,Z 442.218,A -85,B 0,C 180,E1 -22723.283,E2 -22723.283} C_VEL
LIN {X 0,Y 215.491,Z 443.808,A -85,B 0,C 180,E1 -22723.529,E2 -22723.529} C_VEL
LIN {X 0,Y 212.017,Z 498.196,A -85,B 0,C 180,E1 -22725.137,E2 -22725.137} C_VEL
LIN {X 0,Y 210.654,Z 512.556,A -85,B 0,C 180,E1 -22725.695,E2 -22725.695} C_VEL
LIN {X 0,Y 208.267,Z 527.038,A -85,B 0,C 180,E1 -22726.568,E2 -22726.568} C_VEL
LIN {X 0,Y 205.225,Z 540.863,A -85,B 0,C 180,E1 -22727.778,E2 -22727.778} C_VEL
LIN {X 0,Y 201.795,Z 553.308,A -85,B 0,C 180,E1 -22729.235,E2 -22729.235} C_VEL
LIN {X 0,Y 197.963,Z 565.033,A -85,B 0,C 180,E1 -22731.009,E2 -22731.009} C_VEL
LIN {X 0,Y 193.619,Z 576.988,A -85,B 0,C 180,E1 -22733.359,E2 -22733.359} C_VEL
LIN {X 0,Y 188.87,Z 588.002,A -85,B 0,C 180,E1 -22736.075,E2 -22736.075} C_VEL
LIN {X 0,Y 184.494,Z 597.424,A -85,B 0,C 180,E1 -22739.056,E2 -22739.056} C_VEL
LIN {X 0,Y 179.975,Z 606.397,A -85,B 0,C 180,E1 -22742.692,E2 -22742.692} C_VEL
LIN {X 0,Y 176.293,Z 613.65,A -85,B 0,C 180,E1 -22746.51,E2 -22746.51} C_VEL
LIN {X 0,Y 173.837,Z 618.735,A -85,B 0,C 180,E1 -22749.905,E2 -22749.905} C_VEL
LIN {X 0,Y 171.179,Z 623.984,A -85,B 0,C 180,E1 -22754.526,E2 -22754.526} C_VEL
LIN {X 0,Y 169.974,Z 626.929,A -85,B 0,C 180,E1 -22758.073,E2 -22758.073} C_VEL
LIN {X 0,Y 169.044,Z 629.617,A -85,B 0,C 180,E1 -22762.839,E2 -22762.839} C_VEL
LIN {X 0,Y 168.782,Z 630.943,A -85,B 0,C 180,E1 -22767.617,E2 -22767.617} C_VEL
LIN {X 0,Y 168.872,Z 631.104,A -85,B 0,C 180,E1 -22770.004,E2 -22770.004} C_VEL
LIN {X 0,Y 168.86,Z 630.422,A -85,B 0,C 180,E1 -22774.778,E2 -22774.778} C_VEL
LIN {X 0,Y 169.411,Z 628.395,A -85,B 0,C 180,E1 -22779.555,E2 -22779.555} C_VEL
LIN {X 0,Y 170.72,Z 624.98,A -85,B 0,C 180,E1 -22784.304,E2 -22784.304} C_VEL
LIN {X 0,Y 173.131,Z 620.078,A -85,B 0,C 180,E1 -22788.954,E2 -22788.954} C_VEL
LIN {X 0,Y 176.383,Z 613.531,A -85,B 0,C 180,E1 -22793.485,E2 -22793.485} C_VEL
LIN {X 0,Y 176.825,Z 612.77,A -85,B 0,C 180,E1 -22793.982,E2 -22793.982} C_VEL
LIN {X 0,Y 181.239,Z 611.954,A -85,B 0,C 180,E1 -22797.735,E2 -22797.735} C_VEL
LIN {X 0,Y 187.438,Z 609.903,A -85,B 0,C 180,E1 -22801.667,E2 -22801.667} C_VEL
LIN {X 0,Y 194.808,Z 606.629,A -85,B 0,C 180,E1 -22805.259,E2 -22805.259} C_VEL
LIN {X 0,Y 203.301,Z 602.045,A -85,B 0,C 180,E1 -22808.484,E2 -22808.484} C_VEL
LIN {X 0,Y 212.713,Z 596.024,A -85,B 0,C 180,E1 -22811.364,E2 -22811.364} C_VEL
LIN {X 0,Y 222.948,Z 588.467,A -85,B 0,C 180,E1 -22813.911,E2 -22813.911} C_VEL
LIN {X 0,Y 232.459,Z 580.405,A -85,B 0,C 180,E1 -22815.873,E2 -22815.873} C_VEL
LIN {X 0,Y 236.043,Z 577.088,A -85,B 0,C 180,E1 -22816.513,E2 -22816.513} C_VEL
LIN {X 0,Y 236.639,Z 576.502,A -85,B 0,C 180,E1 -22816.915,E2 -22816.915} C_VEL
LIN {X 0,Y 227.278,Z 584.501,A -85,B 0,C 180,E1 -22818.921,E2 -22818.921} C_VEL
LIN {X 0,Y 218.357,Z 590.965,A -85,B 0,C 180,E1 -22821.125,E2 -22821.125} C_VEL
LIN {X 0,Y 209.438,Z 596.354,A -85,B 0,C 180,E1 -22823.77,E2 -22823.77} C_VEL
LIN {X 0,Y 202.336,Z 599.817,A -85,B 0,C 180,E1 -22826.238,E2 -22826.238} C_VEL
LIN {X 0,Y 194.342,Z 602.727,A -85,B 0,C 180,E1 -22829.584,E2 -22829.584} C_VEL
LIN {X 0,Y 187.285,Z 604.254,A -85,B 0,C 180,E1 -22833.237,E2 -22833.237} C_VEL
LIN {X 0,Y 181.323,Z 604.395,A -85,B 0,C 180,E1 -22837.195,E2 -22837.195} C_VEL
LIN {X 0,Y 178.712,Z 603.928,A -85,B 0,C 180,E1 -22839.272,E2 -22839.272} C_VEL
LIN {X 0,Y 174.801,Z 601.969,A -85,B 0,C 180,E1 -22843.654,E2 -22843.654} C_VEL
LIN {X 0,Y 171.937,Z 598.624,A -85,B 0,C 180,E1 -22848.207,E2 -22848.207} C_VEL
LIN {X 0,Y 170.253,Z 593.717,A -85,B 0,C 180,E1 -22852.886,E2 -22852.886} C_VEL
LIN {X 0,Y 169.872,Z 588.965,A -85,B 0,C 180,E1 -22856.442,E2 -22856.442} C_VEL
LIN {X 0,Y 169.776,Z 581.95,A -85,B 0,C 180,E1 -22860.593,E2 -22860.593} C_VEL
LIN {X 0,Y 169.981,Z 574.401,A -85,B 0,C 180,E1 -22864.149,E2 -22864.149} C_VEL
LIN {X 0,Y 170.458,Z 565.072,A -85,B 0,C 180,E1 -22867.701,E2 -22867.701} C_VEL
LIN {X 0,Y 171.152,Z 554.533,A -85,B 0,C 180,E1 -22870.948,E2 -22870.948} C_VEL
LIN {X 0,Y 172.116,Z 542.715,A -85,B 0,C 180,E1 -22873.88,E2 -22873.88} C_VEL
LIN {X 0,Y 173.054,Z 531.008,A -85,B 0,C 180,E1 -22876.213,E2 -22876.213} C_VEL
LIN {X 0,Y 174.067,Z 517.105,A -85,B 0,C 180,E1 -22878.387,E2 -22878.387} C_VEL
LIN {X 0,Y 175.109,Z 501.66,A -85,B 0,C 180,E1 -22880.177,E2 -22880.177} C_VEL
LIN {X 0,Y 176.367,Z 474.492,A -85,B 0,C 180,E1 -22882.322,E2 -22882.322} C_VEL
LIN {X 0,Y 179.186,Z 417.816,A -85,B 0,C 180,E1 -22886.48,E2 -22886.48} C_VEL
LIN {X 0,Y 178.712,Z 413.133,A -85,B 0,C 180,E1 -22886.866,E2 -22886.866} C_VEL
LIN {X 0,Y 179.195,Z 414.61,A -85,B 0,C 180,E1 -22887.297,E2 -22887.297} C_VEL
LIN {X 0,Y 180.345,Z 414.356,A -85,B 0,C 180,E1 -22887.978,E2 -22887.978} C_VEL
LIN {X 0,Y 181.764,Z 412.027,A -85,B 0,C 180,E1 -22888.624,E2 -22888.624} C_VEL
LIN {X 0,Y 183.727,Z 406.656,A -85,B 0,C 180,E1 -22889.312,E2 -22889.312} C_VEL
LIN {X 0,Y 185.159,Z 401.729,A -85,B 0,C 180,E1 -22889.718,E2 -22889.718} C_VEL
LIN {X 0,Y 187.11,Z 400.004,A -85,B 0,C 180,E1 -22890.625,E2 -22890.625} C_VEL
LIN {X 0,Y 188.708,Z 397.598,A -85,B 0,C 180,E1 -22891.265,E2 -22891.265} C_VEL
LIN {X 0,Y 190.943,Z 397.36,A -85,B 0,C 180,E1 -22892.339,E2 -22892.339} C_VEL
LIN {X 0,Y 193.425,Z 400.775,A -85,B 0,C 180,E1 -22893.712,E2 -22893.712} C_VEL
LIN {X 0,Y 197.937,Z 407.097,A -85,B 0,C 180,E1 -22896.013,E2 -22896.013} C_VEL
LIN {X 0,Y 204.515,Z 417.405,A -85,B 0,C 180,E1 -22899.051,E2 -22899.051} C_VEL
LIN {X 0,Y 210.041,Z 428.486,A -85,B 0,C 180,E1 -22901.444,E2 -22901.444} C_VEL
LIN {X 0,Y 214.324,Z 438.417,A -85,B 0,C 180,E1 -22903.208,E2 -22903.208} C_VEL
LIN {X 0,Y 215.455,Z 441.327,A -85,B 0,C 180,E1 -22903.666,E2 -22903.666} C_VEL
LIN {X 0,Y 212.935,Z 481.163,A -85,B 0,C 180,E1 -22904.85,E2 -22904.85} C_VEL
LIN {X 0,Y 211.234,Z 504.733,A -85,B 0,C 180,E1 -22905.608,E2 -22905.608} C_VEL
LIN {X 0,Y 209.493,Z 517.884,A -85,B 0,C 180,E1 -22906.298,E2 -22906.298} C_VEL
LIN {X 0,Y 206.804,Z 531.783,A -85,B 0,C 180,E1 -22907.344,E2 -22907.344} C_VEL
LIN {X 0,Y 203.643,Z 544.711,A -85,B 0,C 180,E1 -22908.694,E2 -22908.694} C_VEL
LIN {X 0,Y 199.866,Z 557.253,A -85,B 0,C 180,E1 -22910.403,E2 -22910.403} C_VEL
LIN {X 0,Y 195.573,Z 569.863,A -85,B 0,C 180,E1 -22912.666,E2 -22912.666} C_VEL
LIN {X 0,Y 190.972,Z 581.104,A -85,B 0,C 180,E1 -22915.217,E2 -22915.217} C_VEL
LIN {X 0,Y 186.416,Z 591.152,A -85,B 0,C 180,E1 -22918.139,E2 -22918.139} C_VEL
LIN {X 0,Y 182.35,Z 599.494,A -85,B 0,C 180,E1 -22921.196,E2 -22921.196} C_VEL
LIN {X 0,Y 178.854,Z 606.454,A -85,B 0,C 180,E1 -22924.387,E2 -22924.387} C_VEL
LIN {X 0,Y 175.986,Z 612.199,A -85,B 0,C 180,E1 -22927.701,E2 -22927.701} C_VEL
LIN {X 0,Y 173.513,Z 616.919,A -85,B 0,C 180,E1 -22931.089,E2 -22931.089} C_VEL
LIN {X 0,Y 171.094,Z 621.803,A -85,B 0,C 180,E1 -22935.728,E2 -22935.728} C_VEL
LIN {X 0,Y 169.643,Z 625.2,A -85,B 0,C 180,E1 -22940.458,E2 -22940.458} C_VEL
LIN {X 0,Y 168.953,Z 627.217,A -85,B 0,C 180,E1 -22945.224,E2 -22945.224} C_VEL
LIN {X 0,Y 168.882,Z 627.903,A -85,B 0,C 180,E1 -22949.996,E2 -22949.996} C_VEL
LIN {X 0,Y 168.951,Z 627.272,A -85,B 0,C 180,E1 -22954.769,E2 -22954.769} C_VEL
LIN {X 0,Y 169.254,Z 626.458,A -85,B 0,C 180,E1 -22957.152,E2 -22957.152} C_VEL
LIN {X 0,Y 170.239,Z 623.808,A -85,B 0,C 180,E1 -22961.909,E2 -22961.909} C_VEL
LIN {X 0,Y 172.077,Z 619.73,A -85,B 0,C 180,E1 -22966.608,E2 -22966.608} C_VEL
LIN {X 0,Y 175.06,Z 614.096,A -85,B 0,C 180,E1 -22971.177,E2 -22971.177} C_VEL
LIN {X 0,Y 177.702,Z 608.726,A -85,B 0,C 180,E1 -22974.544,E2 -22974.544} C_VEL
LIN {X 0,Y 181.65,Z 601.064,A -85,B 0,C 180,E1 -22978.287,E2 -22978.287} C_VEL
LIN {X 0,Y 185.638,Z 593.045,A -85,B 0,C 180,E1 -22981.365,E2 -22981.365} C_VEL
LIN {X 0,Y 190.116,Z 583.374,A -85,B 0,C 180,E1 -22984.311,E2 -22984.311} C_VEL
LIN {X 0,Y 194.658,Z 572.637,A -85,B 0,C 180,E1 -22986.882,E2 -22986.882} C_VEL
LIN {X 0,Y 198.555,Z 561.652,A -85,B 0,C 180,E1 -22989.015,E2 -22989.015} C_VEL
LIN {X 0,Y 202.07,Z 550.625,A -85,B 0,C 180,E1 -22990.697,E2 -22990.697} C_VEL
LIN {X 0,Y 205.451,Z 538.251,A -85,B 0,C 180,E1 -22992.165,E2 -22992.165} C_VEL
LIN {X 0,Y 208.414,Z 524.522,A -85,B 0,C 180,E1 -22993.394,E2 -22993.394} C_VEL
LIN {X 0,Y 210.74,Z 510.196,A -85,B 0,C 180,E1 -22994.282,E2 -22994.282} C_VEL
LIN {X 0,Y 212.129,Z 496.077,A -85,B 0,C 180,E1 -22994.843,E2 -22994.843} C_VEL
LIN {X 0,Y 215.675,Z 441.615,A -85,B 0,C 180,E1 -22996.435,E2 -22996.435} C_VEL
LIN {X 0,Y 210.619,Z 429.575,A -85,B 0,C 180,E1 -22998.507,E2 -22998.507} C_VEL
LIN {X 0,Y 204.502,Z 417.28,A -85,B 0,C 180,E1 -23001.157,E2 -23001.157} C_VEL
LIN {X 0,Y 197.586,Z 406.516,A -85,B 0,C 180,E1 -23004.377,E2 -23004.377} C_VEL
LIN {X 0,Y 191.731,Z 398.282,A -85,B 0,C 180,E1 -23007.459,E2 -23007.459} C_VEL
LIN {X 0,Y 188.05,Z 393.446,A -85,B 0,C 180,E1 -23009.622,E2 -23009.622} C_VEL
LIN {X 0,Y 185.358,Z 389.761,A -85,B 0,C 180,E1 -23011.366,E2 -23011.366} C_VEL
LIN {X 0,Y 182.143,Z 386.293,A -85,B 0,C 180,E1 -23013.581,E2 -23013.581} C_VEL
LIN {X 0,Y 180.937,Z 384.191,A -85,B 0,C 180,E1 -23014.552,E2 -23014.552} C_VEL
LIN {X 0,Y 178.229,Z 381.98,A -85,B 0,C 180,E1 -23016.671,E2 -23016.671} C_VEL
LIN {X 0,Y 176.596,Z 379.066,A -85,B 0,C 180,E1 -23018.246,E2 -23018.246} C_VEL
LIN {X 0,Y 176.17,Z 378.564,A -85,B 0,C 180,E1 -23018.652,E2 -23018.652} C_VEL
LIN {X 0,Y 173.515,Z 376.819,A -85,B 0,C 180,E1 -23021.246,E2 -23021.246} C_VEL
LIN {X 0,Y 171.974,Z 374.528,A -85,B 0,C 180,E1 -23023.148,E2 -23023.148} C_VEL
LIN {X 0,Y 171.547,Z 372.732,A -85,B 0,C 180,E1 -23023.946,E2 -23023.946} C_VEL
LIN {X 0,Y 171.755,Z 372.716,A -85,B 0,C 180,E1 -23029.105,E2 -23029.105} C_VEL
LIN {X 0,Y 171.845,Z 372.704,A -85,B 0,C 180,E1 -23032.952,E2 -23032.952} C_VEL
LIN {X 0,Y 172.061,Z 372.678,A -85,B 0,C 180,E1 -23037.659,E2 -23037.659} C_VEL
LIN {X 0,Y 172.296,Z 372.636,A -85,B 0,C 180,E1 -23040,E2 -23040} C_VEL
LIN {X 0,Y 171.77,Z 372.703,A -85,B 0,C 180,E1 -23044.694,E2 -23044.694} C_VEL
LIN {X 0,Y 171.83,Z 372.697,A -85,B 0,C 180,E1 -23049.416,E2 -23049.416} C_VEL
LIN {X 0,Y 171.541,Z 372.735,A -85,B 0,C 180,E1 -23055.901,E2 -23055.901} C_VEL
LIN {X 0,Y 172.398,Z 375.401,A -85,B 0,C 180,E1 -23057.344,E2 -23057.344} C_VEL
LIN {X 0,Y 174.819,Z 377.941,A -85,B 0,C 180,E1 -23060.021,E2 -23060.021} C_VEL
LIN {X 0,Y 176.542,Z 378.93,A -85,B 0,C 180,E1 -23061.607,E2 -23061.607} C_VEL
LIN {X 0,Y 178.056,Z 381.81,A -85,B 0,C 180,E1 -23063.094,E2 -23063.094} C_VEL
LIN {X 0,Y 181.224,Z 384.709,A -85,B 0,C 180,E1 -23065.597,E2 -23065.597} C_VEL
LIN {X 0,Y 183.551,Z 388.074,A -85,B 0,C 180,E1 -23067.353,E2 -23067.353} C_VEL
LIN {X 0,Y 185.433,Z 389.894,A -85,B 0,C 180,E1 -23068.599,E2 -23068.599} C_VEL
LIN {X 0,Y 188.058,Z 393.51,A -85,B 0,C 180,E1 -23070.299,E2 -23070.299} C_VEL
LIN {X 0,Y 189.348,Z 395.111,A -85,B 0,C 180,E1 -23071.075,E2 -23071.075} C_VEL
LIN {X 0,Y 193.245,Z 400.45,A -85,B 0,C 180,E1 -23073.294,E2 -23073.294} C_VEL
LIN {X 0,Y 196.456,Z 404.999,A -85,B 0,C 180,E1 -23074.977,E2 -23074.977} C_VEL
LIN {X 0,Y 198.814,Z 408.828,A -85,B 0,C 180,E1 -23076.165,E2 -23076.165} C_VEL
LIN {X 0,Y 203.636,Z 417.531,A -85,B 0,C 180,E1 -23078.465,E2 -23078.465} C_VEL
LIN {X 0,Y 209.232,Z 428.822,A -85,B 0,C 180,E1 -23080.934,E2 -23080.934} C_VEL
LIN {X 0,Y 213.747,Z 439.308,A -85,B 0,C 180,E1 -23082.818,E2 -23082.818} C_VEL
LIN {X 0,Y 214.883,Z 442.218,A -85,B 0,C 180,E1 -23083.283,E2 -23083.283} C_VEL
LIN {X 0,Y 215.142,Z 444.608,A -85,B 0,C 180,E1 -23083.47,E2 -23083.47} C_VEL
LIN {X 0,Y 214.426,Z 448.428,A -85,B 0,C 180,E1 -23083.45,E2 -23083.45} C_VEL
LIN {X 0,Y 210.297,Z 458.583,A -85,B 0,C 180,E1 -23082.753,E2 -23082.753} C_VEL
LIN {X 0,Y 209.546,Z 462.02,A -85,B 0,C 180,E1 -23082.701,E2 -23082.701} C_VEL
LIN {X 0,Y 209.494,Z 462.719,A -85,B 0,C 180,E1 -23082.721,E2 -23082.721} C_VEL
LIN {X 0,Y 206.42,Z 505.65,A -85,B 0,C 180,E1 -23084.006,E2 -23084.006} C_VEL
LIN {X 0,Y 204.44,Z 520.408,A -85,B 0,C 180,E1 -23084.762,E2 -23084.762} C_VEL
LIN {X 0,Y 201.873,Z 533.257,A -85,B 0,C 180,E1 -23085.702,E2 -23085.702} C_VEL
LIN {X 0,Y 198.506,Z 546.501,A -85,B 0,C 180,E1 -23087.041,E2 -23087.041} C_VEL
LIN {X 0,Y 194.496,Z 559.265,A -85,B 0,C 180,E1 -23088.746,E2 -23088.746} C_VEL
LIN {X 0,Y 190.322,Z 570.87,A -85,B 0,C 180,E1 -23090.779,E2 -23090.779} C_VEL
LIN {X 0,Y 185.546,Z 582.486,A -85,B 0,C 180,E1 -23093.38,E2 -23093.38} C_VEL
LIN {X 0,Y 180.618,Z 592.874,A -85,B 0,C 180,E1 -23096.33,E2 -23096.33} C_VEL
LIN {X 0,Y 176.29,Z 601.445,A -85,B 0,C 180,E1 -23099.454,E2 -23099.454} C_VEL
LIN {X 0,Y 171.889,Z 609.648,A -85,B 0,C 180,E1 -23103.276,E2 -23103.276} C_VEL
LIN {X 0,Y 168.818,Z 615.547,A -85,B 0,C 180,E1 -23106.815,E2 -23106.815} C_VEL
LIN {X 0,Y 165.642,Z 621.493,A -85,B 0,C 180,E1 -23111.449,E2 -23111.449} C_VEL
LIN {X 0,Y 163.791,Z 624.986,A -85,B 0,C 180,E1 -23115.085,E2 -23115.085} C_VEL
LIN {X 0,Y 162.383,Z 628.379,A -85,B 0,C 180,E1 -23120.035,E2 -23120.035} C_VEL
LIN {X 0,Y 161.762,Z 630.381,A -85,B 0,C 180,E1 -23125.019,E2 -23125.019} C_VEL
LIN {X 0,Y 161.772,Z 631.037,A -85,B 0,C 180,E1 -23130.004,E2 -23130.004} C_VEL
LIN {X 0,Y 161.767,Z 630.354,A -85,B 0,C 180,E1 -23134.988,E2 -23134.988} C_VEL
LIN {X 0,Y 162.39,Z 628.327,A -85,B 0,C 180,E1 -23139.973,E2 -23139.973} C_VEL
LIN {X 0,Y 163.796,Z 624.912,A -85,B 0,C 180,E1 -23144.922,E2 -23144.922} C_VEL
LIN {X 0,Y 166.384,Z 620.009,A -85,B 0,C 180,E1 -23149.754,E2 -23149.754} C_VEL
LIN {X 0,Y 169.843,Z 613.462,A -85,B 0,C 180,E1 -23154.447,E2 -23154.447} C_VEL
LIN {X 0,Y 170.722,Z 612.283,A -85,B 0,C 180,E1 -23155.287,E2 -23155.287} C_VEL
LIN {X 0,Y 174.978,Z 611.837,A -85,B 0,C 180,E1 -23158.818,E2 -23158.818} C_VEL
LIN {X 0,Y 181.462,Z 610.258,A -85,B 0,C 180,E1 -23162.838,E2 -23162.838} C_VEL
LIN {X 0,Y 189.111,Z 607.502,A -85,B 0,C 180,E1 -23166.489,E2 -23166.489} C_VEL
LIN {X 0,Y 197.886,Z 603.487,A -85,B 0,C 180,E1 -23169.741,E2 -23169.741} C_VEL
LIN {X 0,Y 207.616,Z 598.106,A -85,B 0,C 180,E1 -23172.615,E2 -23172.615} C_VEL
LIN {X 0,Y 218.122,Z 591.302,A -85,B 0,C 180,E1 -23175.145,E2 -23175.145} C_VEL
LIN {X 0,Y 224.28,Z 586.806,A -85,B 0,C 180,E1 -23176.418,E2 -23176.418} C_VEL
LIN {X 0,Y 226.39,Z 585.162,A -85,B 0,C 180,E1 -23176.925,E2 -23176.925} C_VEL
LIN {X 0,Y 215.752,Z 592.349,A -85,B 0,C 180,E1 -23179.346,E2 -23179.346} C_VEL
LIN {X 0,Y 208.218,Z 596.555,A -85,B 0,C 180,E1 -23181.36,E2 -23181.36} C_VEL
LIN {X 0,Y 199.662,Z 600.45,A -85,B 0,C 180,E1 -23184.06,E2 -23184.06} C_VEL
LIN {X 0,Y 192.371,Z 602.96,A -85,B 0,C 180,E1 -23186.77,E2 -23186.77} C_VEL
LIN {X 0,Y 184.55,Z 604.643,A -85,B 0,C 180,E1 -23190.326,E2 -23190.326} C_VEL
LIN {X 0,Y 177.775,Z 604.984,A -85,B 0,C 180,E1 -23194.223,E2 -23194.223} C_VEL
LIN {X 0,Y 172.093,Z 603.981,A -85,B 0,C 180,E1 -23198.436,E2 -23198.436} C_VEL
LIN {X 0,Y 168.005,Z 601.594,A -85,B 0,C 180,E1 -23202.973,E2 -23202.973} C_VEL
LIN {X 0,Y 165.052,Z 597.813,A -85,B 0,C 180,E1 -23207.708,E2 -23207.708} C_VEL
LIN {X 0,Y 163.324,Z 592.533,A -85,B 0,C 180,E1 -23212.583,E2 -23212.583} C_VEL
LIN {X 0,Y 162.958,Z 587.45,A -85,B 0,C 180,E1 -23216.291,E2 -23216.291} C_VEL
LIN {X 0,Y 162.84,Z 581.163,A -85,B 0,C 180,E1 -23220,E2 -23220} C_VEL
LIN {X 0,Y 163.062,Z 573.436,A -85,B 0,C 180,E1 -23223.707,E2 -23223.707} C_VEL
LIN {X 0,Y 163.422,Z 565.677,A -85,B 0,C 180,E1 -23226.772,E2 -23226.772} C_VEL
LIN {X 0,Y 164.067,Z 555.24,A -85,B 0,C 180,E1 -23230.178,E2 -23230.178} C_VEL
LIN {X 0,Y 164.983,Z 543.613,A -85,B 0,C 180,E1 -23233.236,E2 -23233.236} C_VEL
LIN {X 0,Y 165.92,Z 532.169,A -85,B 0,C 180,E1 -23235.666,E2 -23235.666} C_VEL
LIN {X 0,Y 166.973,Z 517.586,A -85,B 0,C 180,E1 -23238.085,E2 -23238.085} C_VEL
LIN {X 0,Y 167.976,Z 502.329,A -85,B 0,C 180,E1 -23239.953,E2 -23239.953} C_VEL
LIN {X 0,Y 169.3,Z 473.655,A -85,B 0,C 180,E1 -23242.34,E2 -23242.34} C_VEL
LIN {X 0,Y 170.587,Z 446.975,A -85,B 0,C 180,E1 -23244.437,E2 -23244.437} C_VEL
LIN {X 0,Y 170.833,Z 449.568,A -85,B 0,C 180,E1 -23244.891,E2 -23244.891} C_VEL
LIN {X 0,Y 171.531,Z 449.547,A -85,B 0,C 180,E1 -23245.39,E2 -23245.39} C_VEL
LIN {X 0,Y 172.594,Z 447.731,A -85,B 0,C 180,E1 -23245.957,E2 -23245.957} C_VEL
LIN {X 0,Y 174.541,Z 442.44,A -85,B 0,C 180,E1 -23246.774,E2 -23246.774} C_VEL
LIN {X 0,Y 177.957,Z 430.479,A -85,B 0,C 180,E1 -23247.888,E2 -23247.888} C_VEL
LIN {X 0,Y 180.252,Z 421.404,A -85,B 0,C 180,E1 -23248.506,E2 -23248.506} C_VEL
LIN {X 0,Y 182.134,Z 419.586,A -85,B 0,C 180,E1 -23249.438,E2 -23249.438} C_VEL
LIN {X 0,Y 184.153,Z 416.158,A -85,B 0,C 180,E1 -23250.278,E2 -23250.278} C_VEL
LIN {X 0,Y 186.46,Z 410.157,A -85,B 0,C 180,E1 -23251.037,E2 -23251.037} C_VEL
LIN {X 0,Y 187.495,Z 406.951,A -85,B 0,C 180,E1 -23251.33,E2 -23251.33} C_VEL
LIN {X 0,Y 189.34,Z 404.845,A -85,B 0,C 180,E1 -23252.091,E2 -23252.091} C_VEL
LIN {X 0,Y 193.745,Z 411.056,A -85,B 0,C 180,E1 -23254.519,E2 -23254.519} C_VEL
LIN {X 0,Y 199.894,Z 420.706,A -85,B 0,C 180,E1 -23257.574,E2 -23257.574} C_VEL
LIN {X 0,Y 203.541,Z 427.629,A -85,B 0,C 180,E1 -23259.273,E2 -23259.273} C_VEL
LIN {X 0,Y 209.003,Z 439.783,A -85,B 0,C 180,E1 -23261.696,E2 -23261.696} C_VEL
LIN {X 0,Y 210.453,Z 443.588,A -85,B 0,C 180,E1 -23262.328,E2 -23262.328} C_VEL
LIN {X 0,Y 208.006,Z 481.15,A -85,B 0,C 180,E1 -23263.463,E2 -23263.463} C_VEL
LIN {X 0,Y 206.219,Z 504.909,A -85,B 0,C 180,E1 -23264.235,E2 -23264.235} C_VEL
LIN {X 0,Y 204.419,Z 517.961,A -85,B 0,C 180,E1 -23264.922,E2 -23264.922} C_VEL
LIN {X 0,Y 201.637,Z 531.858,A -85,B 0,C 180,E1 -23265.976,E2 -23265.976} C_VEL
LIN {X 0,Y 198.368,Z 544.784,A -85,B 0,C 180,E1 -23267.342,E2 -23267.342} C_VEL
LIN {X 0,Y 194.438,Z 557.325,A -85,B 0,C 180,E1 -23269.067,E2 -23269.067} C_VEL
LIN {X 0,Y 190.39,Z 568.762,A -85,B 0,C 180,E1 -23271.128,E2 -23271.128} C_VEL
LIN {X 0,Y 186.05,Z 579.259,A -85,B 0,C 180,E1 -23273.487,E2 -23273.487} C_VEL
LIN {X 0,Y 181.909,Z 588.062,A -85,B 0,C 180,E1 -23275.927,E2 -23275.927} C_VEL
LIN {X 0,Y 177.551,Z 596.934,A -85,B 0,C 180,E1 -23279.027,E2 -23279.027} C_VEL
LIN {X 0,Y 173.592,Z 604.314,A -85,B 0,C 180,E1 -23282.248,E2 -23282.248} C_VEL
LIN {X 0,Y 170.392,Z 610.464,A -85,B 0,C 180,E1 -23285.637,E2 -23285.637} C_VEL
LIN {X 0,Y 167.638,Z 615.549,A -85,B 0,C 180,E1 -23289.12,E2 -23289.12} C_VEL
LIN {X 0,Y 164.712,Z 620.812,A -85,B 0,C 180,E1 -23293.895,E2 -23293.895} C_VEL
LIN {X 0,Y 163.289,Z 623.747,A -85,B 0,C 180,E1 -23297.569,E2 -23297.569} C_VEL
LIN {X 0,Y 162.197,Z 626.444,A -85,B 0,C 180,E1 -23302.527,E2 -23302.527} C_VEL
LIN {X 0,Y 161.763,Z 627.833,A -85,B 0,C 180,E1 -23307.814,E2 -23307.814} C_VEL
LIN {X 0,Y 161.765,Z 627.843,A -85,B 0,C 180,E1 -23312.206,E2 -23312.206} C_VEL
LIN {X 0,Y 162.191,Z 626.525,A -85,B 0,C 180,E1 -23317.465,E2 -23317.465} C_VEL
LIN {X 0,Y 163.264,Z 623.875,A -85,B 0,C 180,E1 -23322.425,E2 -23322.425} C_VEL
LIN {X 0,Y 165.253,Z 619.796,A -85,B 0,C 180,E1 -23327.316,E2 -23327.316} C_VEL
LIN {X 0,Y 168.406,Z 614.163,A -85,B 0,C 180,E1 -23332.057,E2 -23332.057} C_VEL
LIN {X 0,Y 171.682,Z 608.013,A -85,B 0,C 180,E1 -23335.97,E2 -23335.97} C_VEL
LIN {X 0,Y 176.072,Z 599.901,A -85,B 0,C 180,E1 -23339.926,E2 -23339.926} C_VEL
LIN {X 0,Y 180.35,Z 591.627,A -85,B 0,C 180,E1 -23343.059,E2 -23343.059} C_VEL
LIN {X 0,Y 185.093,Z 581.659,A -85,B 0,C 180,E1 -23346.049,E2 -23346.049} C_VEL
LIN {X 0,Y 189.88,Z 570.557,A -85,B 0,C 180,E1 -23348.648,E2 -23348.648} C_VEL
LIN {X 0,Y 193.881,Z 559.508,A -85,B 0,C 180,E1 -23350.724,E2 -23350.724} C_VEL
LIN {X 0,Y 197.706,Z 547.501,A -85,B 0,C 180,E1 -23352.481,E2 -23352.481} C_VEL
LIN {X 0,Y 201.296,Z 534.196,A -85,B 0,C 180,E1 -23353.936,E2 -23353.936} C_VEL
LIN {X 0,Y 204.143,Z 520.355,A -85,B 0,C 180,E1 -23355.06,E2 -23355.06} C_VEL
LIN {X 0,Y 206.296,Z 505.335,A -85,B 0,C 180,E1 -23355.891,E2 -23355.891} C_VEL
LIN {X 0,Y 208.097,Z 483.132,A -85,B 0,C 180,E1 -23356.594,E2 -23356.594} C_VEL
LIN {X 0,Y 210.592,Z 443.693,A -85,B 0,C 180,E1 -23357.808,E2 -23357.808} C_VEL
LIN {X 0,Y 205.973,Z 432.701,A -85,B 0,C 180,E1 -23359.826,E2 -23359.826} C_VEL
LIN {X 0,Y 200.752,Z 422.041,A -85,B 0,C 180,E1 -23362.235,E2 -23362.235} C_VEL
LIN {X 0,Y 194.538,Z 412.114,A -85,B 0,C 180,E1 -23365.294,E2 -23365.294} C_VEL
LIN {X 0,Y 188.83,Z 403.938,A -85,B 0,C 180,E1 -23368.463,E2 -23368.463} C_VEL
LIN {X 0,Y 185.738,Z 399.713,A -85,B 0,C 180,E1 -23370.379,E2 -23370.379} C_VEL
LIN {X 0,Y 182.618,Z 395.577,A -85,B 0,C 180,E1 -23372.495,E2 -23372.495} C_VEL
LIN {X 0,Y 179.773,Z 392.154,A -85,B 0,C 180,E1 -23374.606,E2 -23374.606} C_VEL
LIN {X 0,Y 178.83,Z 390.699,A -85,B 0,C 180,E1 -23375.389,E2 -23375.389} C_VEL
LIN {X 0,Y 175.926,Z 387.821,A -85,B 0,C 180,E1 -23377.851,E2 -23377.851} C_VEL
LIN {X 0,Y 174.615,Z 385.392,A -85,B 0,C 180,E1 -23379.21,E2 -23379.21} C_VEL
LIN {X 0,Y 171.921,Z 383.38,A -85,B 0,C 180,E1 -23381.992,E2 -23381.992} C_VEL
LIN {X 0,Y 170.313,Z 380.77,A -85,B 0,C 180,E1 -23384.134,E2 -23384.134} C_VEL
LIN {X 0,Y 169.969,Z 379.698,A -85,B 0,C 180,E1 -23384.716,E2 -23384.716} C_VEL
LIN {X 0,Y 167.131,Z 378.1,A -85,B 0,C 180,E1 -23389.188,E2 -23389.188} C_VEL
LIN {X 0,Y 164.984,Z 374.532,A -85,B 0,C 180,E1 -23396.183,E2 -23396.183} C_VEL
LIN {X 0,Y 164.935,Z 373.564,A -85,B 0,C 180,E1 -23397.252,E2 -23397.252} C_VEL
LIN {X 0,Y 165.261,Z 373.513,A -85,B 0,C 180,E1 -23400,E2 -23400} C_VEL
LIN {X 0,Y 164.939,Z 373.763,A -85,B 0,C 180,E1 -23402.9,E2 -23402.9} C_VEL
LIN {X 0,Y 165.205,Z 375.424,A -85,B 0,C 180,E1 -23405.186,E2 -23405.186} C_VEL
LIN {X 0,Y 168.969,Z 379.351,A -85,B 0,C 180,E1 -23413.837,E2 -23413.837} C_VEL
LIN {X 0,Y 170.02,Z 379.832,A -85,B 0,C 180,E1 -23415.279,E2 -23415.279} C_VEL
LIN {X 0,Y 171.179,Z 382.46,A -85,B 0,C 180,E1 -23417.009,E2 -23417.009} C_VEL
LIN {X 0,Y 173.6,Z 384.881,A -85,B 0,C 180,E1 -23419.737,E2 -23419.737} C_VEL
LIN {X 0,Y 174.813,Z 385.76,A -85,B 0,C 180,E1 -23420.914,E2 -23420.914} C_VEL
LIN {X 0,Y 176.588,Z 388.731,A -85,B 0,C 180,E1 -23422.678,E2 -23422.678} C_VEL
LIN {X 0,Y 179.218,Z 391.207,A -85,B 0,C 180,E1 -23424.84,E2 -23424.84} C_VEL
LIN {X 0,Y 181.813,Z 394.802,A -85,B 0,C 180,E1 -23426.858,E2 -23426.858} C_VEL
LIN {X 0,Y 183.337,Z 396.513,A -85,B 0,C 180,E1 -23427.922,E2 -23427.922} C_VEL
LIN {X 0,Y 186.994,Z 401.454,A -85,B 0,C 180,E1 -23430.334,E2 -23430.334} C_VEL
LIN {X 0,Y 190.646,Z 406.541,A -85,B 0,C 180,E1 -23432.507,E2 -23432.507} C_VEL
LIN {X 0,Y 194.402,Z 411.971,A -85,B 0,C 180,E1 -23434.55,E2 -23434.55} C_VEL
LIN {X 0,Y 199.874,Z 422.131,A -85,B 0,C 180,E1 -23437.356,E2 -23437.356} C_VEL
LIN {X 0,Y 205.231,Z 433.231,A -85,B 0,C 180,E1 -23439.867,E2 -23439.867} C_VEL
LIN {X 0,Y 209.934,Z 444.584,A -85,B 0,C 180,E1 -23441.95,E2 -23441.95} C_VEL
LIN {X 0,Y 210.492,Z 446,A -85,B 0,C 180,E1 -23442.189,E2 -23442.189} C_VEL
LIN {X 0,Y 209.494,Z 462.719,A -85,B 0,C 180,E1 -23442.721,E2 -23442.721} C_VEL
LIN {X 0,Y 208.726,Z 468.569,A -85,B 0,C 180,E1 -23442.783,E2 -23442.783} C_VEL
LIN {X 0,Y 206.101,Z 478.08,A -85,B 0,C 180,E1 -23442.472,E2 -23442.472} C_VEL
LIN {X 0,Y 203.415,Z 487.593,A -85,B 0,C 180,E1 -23442.133,E2 -23442.133} C_VEL
LIN {X 0,Y 202.543,Z 493.453,A -85,B 0,C 180,E1 -23442.164,E2 -23442.164} C_VEL
LIN {X 0,Y 201.171,Z 509.43,A -85,B 0,C 180,E1 -23442.745,E2 -23442.745} C_VEL
LIN {X 0,Y 198.775,Z 524.159,A -85,B 0,C 180,E1 -23443.552,E2 -23443.552} C_VEL
LIN {X 0,Y 195.77,Z 537.715,A -85,B 0,C 180,E1 -23444.668,E2 -23444.668} C_VEL
LIN {X 0,Y 192.307,Z 549.974,A -85,B 0,C 180,E1 -23446.028,E2 -23446.028} C_VEL
LIN {X 0,Y 188.192,Z 562.047,A -85,B 0,C 180,E1 -23447.767,E2 -23447.767} C_VEL
LIN {X 0,Y 183.706,Z 573.674,A -85,B 0,C 180,E1 -23449.966,E2 -23449.966} C_VEL
LIN {X 0,Y 179,Z 584.307,A -85,B 0,C 180,E1 -23452.519,E2 -23452.519} C_VEL
LIN {X 0,Y 173.904,Z 594.32,A -85,B 0,C 180,E1 -23455.548,E2 -23455.548} C_VEL
LIN {X 0,Y 169.468,Z 602.638,A -85,B 0,C 180,E1 -23458.781,E2 -23458.781} C_VEL
LIN {X 0,Y 164.963,Z 610.591,A -85,B 0,C 180,E1 -23462.747,E2 -23462.747} C_VEL
LIN {X 0,Y 161.407,Z 616.993,A -85,B 0,C 180,E1 -23466.933,E2 -23466.933} C_VEL
LIN {X 0,Y 158.163,Z 622.672,A -85,B 0,C 180,E1 -23471.882,E2 -23471.882} C_VEL
LIN {X 0,Y 156.02,Z 626.795,A -85,B 0,C 180,E1 -23476.988,E2 -23476.988} C_VEL
LIN {X 0,Y 154.929,Z 629.483,A -85,B 0,C 180,E1 -23482.183,E2 -23482.183} C_VEL
LIN {X 0,Y 154.59,Z 630.808,A -85,B 0,C 180,E1 -23487.398,E2 -23487.398} C_VEL
LIN {X 0,Y 154.624,Z 630.936,A -85,B 0,C 180,E1 -23490.604,E2 -23490.604} C_VEL
LIN {X 0,Y 154.696,Z 630.286,A -85,B 0,C 180,E1 -23495.217,E2 -23495.217} C_VEL
LIN {X 0,Y 155.389,Z 628.259,A -85,B 0,C 180,E1 -23500.427,E2 -23500.427} C_VEL
LIN {X 0,Y 156.9,Z 624.843,A -85,B 0,C 180,E1 -23505.594,E2 -23505.594} C_VEL
LIN {X 0,Y 159.662,Z 619.94,A -85,B 0,C 180,E1 -23510.622,E2 -23510.622} C_VEL
LIN {X 0,Y 163.1,Z 613.841,A -85,B 0,C 180,E1 -23515.191,E2 -23515.191} C_VEL
LIN {X 0,Y 164.655,Z 611.645,A -85,B 0,C 180,E1 -23516.63,E2 -23516.63} C_VEL
LIN {X 0,Y 168.794,Z 611.564,A -85,B 0,C 180,E1 -23519.98,E2 -23519.98} C_VEL
LIN {X 0,Y 175.545,Z 610.448,A -85,B 0,C 180,E1 -23524.094,E2 -23524.094} C_VEL
LIN {X 0,Y 183.492,Z 608.19,A -85,B 0,C 180,E1 -23527.797,E2 -23527.797} C_VEL
LIN {X 0,Y 192.567,Z 604.734,A -85,B 0,C 180,E1 -23531.07,E2 -23531.07} C_VEL
LIN {X 0,Y 202.574,Z 600.008,A -85,B 0,C 180,E1 -23533.941,E2 -23533.941} C_VEL
LIN {X 0,Y 213.376,Z 593.904,A -85,B 0,C 180,E1 -23536.44,E2 -23536.44} C_VEL
LIN {X 0,Y 214.521,Z 593.208,A -85,B 0,C 180,E1 -23536.685,E2 -23536.685} C_VEL
LIN {X 0,Y 215.33,Z 592.681,A -85,B 0,C 180,E1 -23537.086,E2 -23537.086} C_VEL
LIN {X 0,Y 205.47,Z 597.782,A -85,B 0,C 180,E1 -23539.467,E2 -23539.467} C_VEL
LIN {X 0,Y 195.647,Z 601.734,A -85,B 0,C 180,E1 -23542.362,E2 -23542.362} C_VEL
LIN {X 0,Y 186.58,Z 604.305,A -85,B 0,C 180,E1 -23545.597,E2 -23545.597} C_VEL
LIN {X 0,Y 178.47,Z 605.478,A -85,B 0,C 180,E1 -23549.208,E2 -23549.208} C_VEL
LIN {X 0,Y 171.437,Z 605.318,A -85,B 0,C 180,E1 -23553.196,E2 -23553.196} C_VEL
LIN {X 0,Y 165.522,Z 603.841,A -85,B 0,C 180,E1 -23557.534,E2 -23557.534} C_VEL
LIN {X 0,Y 161.247,Z 601.057,A -85,B 0,C 180,E1 -23562.236,E2 -23562.236} C_VEL
LIN {X 0,Y 158.188,Z 596.841,A -85,B 0,C 180,E1 -23567.165,E2 -23567.165} C_VEL
LIN {X 0,Y 156.446,Z 591.116,A -85,B 0,C 180,E1 -23572.255,E2 -23572.255} C_VEL
LIN {X 0,Y 156.015,Z 584.697,A -85,B 0,C 180,E1 -23576.772,E2 -23576.772} C_VEL
LIN {X 0,Y 156.024,Z 577.809,A -85,B 0,C 180,E1 -23580.645,E2 -23580.645} C_VEL
LIN {X 0,Y 156.223,Z 570.871,A -85,B 0,C 180,E1 -23583.869,E2 -23583.869} C_VEL
LIN {X 0,Y 156.593,Z 562.564,A -85,B 0,C 180,E1 -23587.09,E2 -23587.09} C_VEL
LIN {X 0,Y 157.222,Z 552.597,A -85,B 0,C 180,E1 -23590.3,E2 -23590.3} C_VEL
LIN {X 0,Y 158.191,Z 540.349,A -85,B 0,C 180,E1 -23593.488,E2 -23593.488} C_VEL
LIN {X 0,Y 159.12,Z 528.143,A -85,B 0,C 180,E1 -23596.025,E2 -23596.025} C_VEL
LIN {X 0,Y 160.078,Z 514.536,A -85,B 0,C 180,E1 -23598.229,E2 -23598.229} C_VEL
LIN {X 0,Y 160.999,Z 500.358,A -85,B 0,C 180,E1 -23599.94,E2 -23599.94} C_VEL
LIN {X 0,Y 161.793,Z 484.704,A -85,B 0,C 180,E1 -23601.334,E2 -23601.334} C_VEL
LIN {X 0,Y 161.717,Z 487.88,A -85,B 0,C 180,E1 -23601.679,E2 -23601.679} C_VEL
LIN {X 0,Y 161.954,Z 488.653,A -85,B 0,C 180,E1 -23601.98,E2 -23601.98} C_VEL
LIN {X 0,Y 162.485,Z 488.341,A -85,B 0,C 180,E1 -23602.406,E2 -23602.406} C_VEL
LIN {X 0,Y 164.384,Z 483.617,A -85,B 0,C 180,E1 -23603.462,E2 -23603.462} C_VEL
LIN {X 0,Y 167.406,Z 473.401,A -85,B 0,C 180,E1 -23604.741,E2 -23604.741} C_VEL
LIN {X 0,Y 171.404,Z 457.338,A -85,B 0,C 180,E1 -23606.04,E2 -23606.04} C_VEL
LIN {X 0,Y 171.653,Z 456.3,A -85,B 0,C 180,E1 -23606.113,E2 -23606.113} C_VEL
LIN {X 0,Y 173.369,Z 454.455,A -85,B 0,C 180,E1 -23607.087,E2 -23607.087} C_VEL
LIN {X 0,Y 175.165,Z 450.931,A -85,B 0,C 180,E1 -23607.917,E2 -23607.917} C_VEL
LIN {X 0,Y 177.611,Z 444.123,A -85,B 0,C 180,E1 -23608.821,E2 -23608.821} C_VEL
LIN {X 0,Y 181.236,Z 431.661,A -85,B 0,C 180,E1 -23609.887,E2 -23609.887} C_VEL
LIN {X 0,Y 182.759,Z 426.294,A -85,B 0,C 180,E1 -23610.302,E2 -23610.302} C_VEL
LIN {X 0,Y 185.374,Z 422.716,A -85,B 0,C 180,E1 -23611.403,E2 -23611.403} C_VEL
LIN {X 0,Y 187.753,Z 417.868,A -85,B 0,C 180,E1 -23612.236,E2 -23612.236} C_VEL
LIN {X 0,Y 189.187,Z 414.237,A -85,B 0,C 180,E1 -23612.671,E2 -23612.671} C_VEL
LIN {X 0,Y 195.142,Z 423.631,A -85,B 0,C 180,E1 -23615.896,E2 -23615.896} C_VEL
LIN {X 0,Y 198.715,Z 430.077,A -85,B 0,C 180,E1 -23617.676,E2 -23617.676} C_VEL
LIN {X 0,Y 204.073,Z 442.028,A -85,B 0,C 180,E1 -23620.233,E2 -23620.233} C_VEL
LIN {X 0,Y 205.591,Z 446.019,A -85,B 0,C 180,E1 -23620.941,E2 -23620.941} C_VEL
LIN {X 0,Y 203.193,Z 481.212,A -85,B 0,C 180,E1 -23622.01,E2 -23622.01} C_VEL
LIN {X 0,Y 201.327,Z 505.089,A -85,B 0,C 180,E1 -23622.793,E2 -23622.793} C_VEL
LIN {X 0,Y 199.468,Z 518.039,A -85,B 0,C 180,E1 -23623.478,E2 -23623.478} C_VEL
LIN {X 0,Y 196.59,Z 531.933,A -85,B 0,C 180,E1 -23624.537,E2 -23624.537} C_VEL
LIN {X 0,Y 193.192,Z 544.857,A -85,B 0,C 180,E1 -23625.91,E2 -23625.91} C_VEL
LIN {X 0,Y 189.118,Z 557.397,A -85,B 0,C 180,E1 -23627.654,E2 -23627.654} C_VEL
LIN {X 0,Y 184.909,Z 568.833,A -85,B 0,C 180,E1 -23629.746,E2 -23629.746} C_VEL
LIN {X 0,Y 180.392,Z 579.329,A -85,B 0,C 180,E1 -23632.145,E2 -23632.145} C_VEL
LIN {X 0,Y 176.062,Z 588.132,A -85,B 0,C 180,E1 -23634.63,E2 -23634.63} C_VEL
LIN {X 0,Y 171.458,Z 597.004,A -85,B 0,C 180,E1 -23637.797,E2 -23637.797} C_VEL
LIN {X 0,Y 166.704,Z 605.497,A -85,B 0,C 180,E1 -23641.684,E2 -23641.684} C_VEL
LIN {X 0,Y 162.87,Z 612.338,A -85,B 0,C 180,E1 -23645.796,E2 -23645.796} C_VEL
LIN {X 0,Y 160.097,Z 617.057,A -85,B 0,C 180,E1 -23649.436,E2 -23649.436} C_VEL
LIN {X 0,Y 157.875,Z 620.88,A -85,B 0,C 180,E1 -23653.177,E2 -23653.177} C_VEL
LIN {X 0,Y 156.339,Z 623.816,A -85,B 0,C 180,E1 -23657.007,E2 -23657.007} C_VEL
LIN {X 0,Y 155.159,Z 626.512,A -85,B 0,C 180,E1 -23662.186,E2 -23662.186} C_VEL
LIN {X 0,Y 154.668,Z 627.86,A -85,B 0,C 180,E1 -23667.392,E2 -23667.392} C_VEL
LIN {X 0,Y 154.656,Z 627.972,A -85,B 0,C 180,E1 -23671.297,E2 -23671.297} C_VEL
LIN {X 0,Y 154.799,Z 627.406,A -85,B 0,C 180,E1 -23675.206,E2 -23675.206} C_VEL
LIN {X 0,Y 155.153,Z 626.592,A -85,B 0,C 180,E1 -23677.806,E2 -23677.806} C_VEL
LIN {X 0,Y 156.315,Z 623.942,A -85,B 0,C 180,E1 -23682.987,E2 -23682.987} C_VEL
LIN {X 0,Y 158.46,Z 619.863,A -85,B 0,C 180,E1 -23688.083,E2 -23688.083} C_VEL
LIN {X 0,Y 161.8,Z 614.229,A -85,B 0,C 180,E1 -23693.008,E2 -23693.008} C_VEL
LIN {X 0,Y 164.915,Z 608.754,A -85,B 0,C 180,E1 -23696.661,E2 -23696.661} C_VEL
LIN {X 0,Y 169.234,Z 601.195,A -85,B 0,C 180,E1 -23700.574,E2 -23700.574} C_VEL
LIN {X 0,Y 173.637,Z 593.175,A -85,B 0,C 180,E1 -23703.812,E2 -23703.812} C_VEL
LIN {X 0,Y 178.521,Z 583.503,A -85,B 0,C 180,E1 -23706.891,E2 -23706.891} C_VEL
LIN {X 0,Y 183.481,Z 572.764,A -85,B 0,C 180,E1 -23709.549,E2 -23709.549} C_VEL
LIN {X 0,Y 187.651,Z 562.002,A -85,B 0,C 180,E1 -23711.704,E2 -23711.704} C_VEL
LIN {X 0,Y 191.535,Z 550.749,A -85,B 0,C 180,E1 -23713.466,E2 -23713.466} C_VEL
LIN {X 0,Y 195.154,Z 538.372,A -85,B 0,C 180,E1 -23714.966,E2 -23714.966} C_VEL
LIN {X 0,Y 198.349,Z 524.639,A -85,B 0,C 180,E1 -23716.209,E2 -23716.209} C_VEL
LIN {X 0,Y 200.845,Z 510.306,A -85,B 0,C 180,E1 -23717.104,E2 -23717.104} C_VEL
LIN {X 0,Y 202.294,Z 496.511,A -85,B 0,C 180,E1 -23717.665,E2 -23717.665} C_VEL
LIN {X 0,Y 205.754,Z 447.138,A -85,B 0,C 180,E1 -23719.138,E2 -23719.138} C_VEL
LIN {X 0,Y 205.487,Z 445.48,A -85,B 0,C 180,E1 -23719.311,E2 -23719.311} C_VEL
LIN {X 0,Y 201.376,Z 435.661,A -85,B 0,C 180,E1 -23721.238,E2 -23721.238} C_VEL
LIN {X 0,Y 197.094,Z 426.809,A -85,B 0,C 180,E1 -23723.345,E2 -23723.345} C_VEL
LIN {X 0,Y 191.428,Z 417.575,A -85,B 0,C 180,E1 -23726.3,E2 -23726.3} C_VEL
LIN {X 0,Y 186.104,Z 409.727,A -85,B 0,C 180,E1 -23729.427,E2 -23729.427} C_VEL
LIN {X 0,Y 183.231,Z 405.684,A -85,B 0,C 180,E1 -23731.309,E2 -23731.309} C_VEL
LIN {X 0,Y 180.343,Z 401.784,A -85,B 0,C 180,E1 -23733.374,E2 -23733.374} C_VEL
LIN {X 0,Y 177.499,Z 398.075,A -85,B 0,C 180,E1 -23735.627,E2 -23735.627} C_VEL
LIN {X 0,Y 176.658,Z 396.99,A -85,B 0,C 180,E1 -23736.345,E2 -23736.345} C_VEL
LIN {X 0,Y 173.97,Z 394,A -85,B 0,C 180,E1 -23738.792,E2 -23738.792} C_VEL
LIN {X 0,Y 172.883,Z 392.087,A -85,B 0,C 180,E1 -23739.97,E2 -23739.97} C_VEL
LIN {X 0,Y 170.247,Z 389.775,A -85,B 0,C 180,E1 -23742.895,E2 -23742.895} C_VEL
LIN {X 0,Y 168.704,Z 387.012,A -85,B 0,C 180,E1 -23745.14,E2 -23745.14} C_VEL
LIN {X 0,Y 168.482,Z 386.538,A -85,B 0,C 180,E1 -23745.506,E2 -23745.506} C_VEL
LIN {X 0,Y 165.756,Z 384.712,A -85,B 0,C 180,E1 -23750.235,E2 -23750.235} C_VEL
LIN {X 0,Y 164.032,Z 381.233,A -85,B 0,C 180,E1 -23756.93,E2 -23756.93} C_VEL
LIN {X 0,Y 164.015,Z 380.697,A -85,B 0,C 180,E1 -23757.544,E2 -23757.544} C_VEL
LIN {X 0,Y 163.974,Z 380.568,A -85,B 0,C 180,E1 -23761.842,E2 -23761.842} C_VEL
LIN {X 0,Y 164.052,Z 381.38,A -85,B 0,C 180,E1 -23763.223,E2 -23763.223} C_VEL
LIN {X 0,Y 166.75,Z 385.647,A -85,B 0,C 180,E1 -23771.695,E2 -23771.695} C_VEL
LIN {X 0,Y 168.626,Z 386.788,A -85,B 0,C 180,E1 -23774.636,E2 -23774.636} C_VEL
LIN {X 0,Y 170.167,Z 389.715,A -85,B 0,C 180,E1 -23776.92,E2 -23776.92} C_VEL
LIN {X 0,Y 172.773,Z 392.039,A -85,B 0,C 180,E1 -23779.836,E2 -23779.836} C_VEL
LIN {X 0,Y 175.586,Z 396.076,A -85,B 0,C 180,E1 -23782.659,E2 -23782.659} C_VEL
LIN {X 0,Y 177.322,Z 397.785,A -85,B 0,C 180,E1 -23784.13,E2 -23784.13} C_VEL
LIN {X 0,Y 180.181,Z 401.589,A -85,B 0,C 180,E1 -23786.417,E2 -23786.417} C_VEL
LIN {X 0,Y 184.546,Z 407.529,A -85,B 0,C 180,E1 -23789.484,E2 -23789.484} C_VEL
LIN {X 0,Y 189.772,Z 414.985,A -85,B 0,C 180,E1 -23792.676,E2 -23792.676} C_VEL
LIN {X 0,Y 193.454,Z 421.357,A -85,B 0,C 180,E1 -23794.744,E2 -23794.744} C_VEL
LIN {X 0,Y 199.086,Z 432.754,A -85,B 0,C 180,E1 -23797.676,E2 -23797.676} C_VEL
LIN {X 0,Y 203.483,Z 442.81,A -85,B 0,C 180,E1 -23799.795,E2 -23799.795} C_VEL
LIN {X 0,Y 205.669,Z 448.518,A -85,B 0,C 180,E1 -23800.819,E2 -23800.819} C_VEL
LIN {X 0,Y 202.543,Z 493.453,A -85,B 0,C 180,E1 -23802.164,E2 -23802.164} C_VEL
LIN {X 0,Y 201.667,Z 499.29,A -85,B 0,C 180,E1 -23802.196,E2 -23802.196} C_VEL
LIN {X 0,Y 198.772,Z 508.737,A -85,B 0,C 180,E1 -23801.936,E2 -23801.936} C_VEL
LIN {X 0,Y 195.506,Z 518.089,A -85,B 0,C 180,E1 -23801.789,E2 -23801.789} C_VEL
LIN {X 0,Y 194.028,Z 523.774,A -85,B 0,C 180,E1 -23802.015,E2 -23802.015} C_VEL
LIN {X 0,Y 190.853,Z 537.655,A -85,B 0,C 180,E1 -23803.154,E2 -23803.154} C_VEL
LIN {X 0,Y 187.263,Z 549.912,A -85,B 0,C 180,E1 -23804.52,E2 -23804.52} C_VEL
LIN {X 0,Y 182.995,Z 561.984,A -85,B 0,C 180,E1 -23806.272,E2 -23806.272} C_VEL
LIN {X 0,Y 178.428,Z 573.389,A -85,B 0,C 180,E1 -23808.45,E2 -23808.45} C_VEL
LIN {X 0,Y 173.409,Z 584.242,A -85,B 0,C 180,E1 -23811.088,E2 -23811.088} C_VEL
LIN {X 0,Y 168.071,Z 594.255,A -85,B 0,C 180,E1 -23814.172,E2 -23814.172} C_VEL
LIN {X 0,Y 163.423,Z 602.572,A -85,B 0,C 180,E1 -23817.487,E2 -23817.487} C_VEL
LIN {X 0,Y 158.632,Z 610.525,A -85,B 0,C 180,E1 -23821.563,E2 -23821.563} C_VEL
LIN {X 0,Y 154.852,Z 616.927,A -85,B 0,C 180,E1 -23825.896,E2 -23825.896} C_VEL
LIN {X 0,Y 151.387,Z 622.606,A -85,B 0,C 180,E1 -23831.041,E2 -23831.041} C_VEL
LIN {X 0,Y 149.069,Z 626.728,A -85,B 0,C 180,E1 -23836.37,E2 -23836.37} C_VEL
LIN {X 0,Y 147.881,Z 629.416,A -85,B 0,C 180,E1 -23841.807,E2 -23841.807} C_VEL
LIN {X 0,Y 147.508,Z 630.741,A -85,B 0,C 180,E1 -23847.273,E2 -23847.273} C_VEL
LIN {X 0,Y 147.588,Z 630.903,A -85,B 0,C 180,E1 -23850.004,E2 -23850.004} C_VEL
LIN {X 0,Y 147.624,Z 630.219,A -85,B 0,C 180,E1 -23855.468,E2 -23855.468} C_VEL
LIN {X 0,Y 148.373,Z 628.191,A -85,B 0,C 180,E1 -23860.926,E2 -23860.926} C_VEL
LIN {X 0,Y 150.033,Z 624.775,A -85,B 0,C 180,E1 -23866.327,E2 -23866.327} C_VEL
LIN {X 0,Y 152.983,Z 619.871,A -85,B 0,C 180,E1 -23871.567,E2 -23871.567} C_VEL
LIN {X 0,Y 157.015,Z 613.325,A -85,B 0,C 180,E1 -23876.594,E2 -23876.594} C_VEL
LIN {X 0,Y 158.678,Z 610.898,A -85,B 0,C 180,E1 -23878.077,E2 -23878.077} C_VEL
LIN {X 0,Y 162.695,Z 611.103,A -85,B 0,C 180,E1 -23881.227,E2 -23881.227} C_VEL
LIN {X 0,Y 169.723,Z 610.45,A -85,B 0,C 180,E1 -23885.435,E2 -23885.435} C_VEL
LIN {X 0,Y 177.949,Z 608.688,A -85,B 0,C 180,E1 -23889.195,E2 -23889.195} C_VEL
LIN {X 0,Y 187.323,Z 605.783,A -85,B 0,C 180,E1 -23892.483,E2 -23892.483} C_VEL
LIN {X 0,Y 197.62,Z 601.682,A -85,B 0,C 180,E1 -23895.342,E2 -23895.342} C_VEL
LIN {X 0,Y 203.053,Z 599.151,A -85,B 0,C 180,E1 -23896.626,E2 -23896.626} C_VEL
LIN {X 0,Y 203.69,Z 598.758,A -85,B 0,C 180,E1 -23897.363,E2 -23897.363} C_VEL
LIN {X 0,Y 195.174,Z 601.966,A -85,B 0,C 180,E1 -23899.597,E2 -23899.597} C_VEL
LIN {X 0,Y 185.41,Z 604.63,A -85,B 0,C 180,E1 -23902.665,E2 -23902.665} C_VEL
LIN {X 0,Y 176.524,Z 605.971,A -85,B 0,C 180,E1 -23906.125,E2 -23906.125} C_VEL
LIN {X 0,Y 168.638,Z 605.981,A -85,B 0,C 180,E1 -23909.994,E2 -23909.994} C_VEL
LIN {X 0,Y 161.945,Z 604.676,A -85,B 0,C 180,E1 -23914.28,E2 -23914.28} C_VEL
LIN {X 0,Y 159.001,Z 603.539,A -85,B 0,C 180,E1 -23916.559,E2 -23916.559} C_VEL
LIN {X 0,Y 154.547,Z 600.318,A -85,B 0,C 180,E1 -23921.439,E2 -23921.439} C_VEL
LIN {X 0,Y 151.384,Z 595.713,A -85,B 0,C 180,E1 -23926.578,E2 -23926.578} C_VEL
LIN {X 0,Y 149.591,Z 589.521,A -85,B 0,C 180,E1 -23931.898,E2 -23931.898} C_VEL
LIN {X 0,Y 149.231,Z 583.758,A -85,B 0,C 180,E1 -23935.949,E2 -23935.949} C_VEL
LIN {X 0,Y 149.183,Z 576.708,A -85,B 0,C 180,E1 -23940,E2 -23940} C_VEL
LIN {X 0,Y 149.412,Z 568.038,A -85,B 0,C 180,E1 -23944.046,E2 -23944.046} C_VEL
LIN {X 0,Y 149.918,Z 558.243,A -85,B 0,C 180,E1 -23947.746,E2 -23947.746} C_VEL
LIN {X 0,Y 150.578,Z 547.574,A -85,B 0,C 180,E1 -23951.036,E2 -23951.036} C_VEL
LIN {X 0,Y 151.549,Z 535.326,A -85,B 0,C 180,E1 -23954.091,E2 -23954.091} C_VEL
LIN {X 0,Y 152.349,Z 523.616,A -85,B 0,C 180,E1 -23956.413,E2 -23956.413} C_VEL
LIN {X 0,Y 152.939,Z 515.575,A -85,B 0,C 180,E1 -23957.725,E2 -23957.725} C_VEL
LIN {X 0,Y 152.853,Z 517.272,A -85,B 0,C 180,E1 -23958.168,E2 -23958.168} C_VEL
LIN {X 0,Y 153.237,Z 517.636,A -85,B 0,C 180,E1 -23958.726,E2 -23958.726} C_VEL
LIN {X 0,Y 154.488,Z 516.412,A -85,B 0,C 180,E1 -23959.69,E2 -23959.69} C_VEL
LIN {X 0,Y 156.52,Z 512.738,A -85,B 0,C 180,E1 -23960.794,E2 -23960.794} C_VEL
LIN {X 0,Y 158.998,Z 506.705,A -85,B 0,C 180,E1 -23961.83,E2 -23961.83} C_VEL
LIN {X 0,Y 161.437,Z 498.672,A -85,B 0,C 180,E1 -23962.719,E2 -23962.719} C_VEL
LIN {X 0,Y 162.32,Z 495.308,A -85,B 0,C 180,E1 -23963.05,E2 -23963.05} C_VEL
LIN {X 0,Y 163.802,Z 493.502,A -85,B 0,C 180,E1 -23964.055,E2 -23964.055} C_VEL
LIN {X 0,Y 165.735,Z 489.231,A -85,B 0,C 180,E1 -23965.091,E2 -23965.091} C_VEL
LIN {X 0,Y 168.11,Z 482.314,A -85,B 0,C 180,E1 -23966.121,E2 -23966.121} C_VEL
LIN {X 0,Y 171.453,Z 470.533,A -85,B 0,C 180,E1 -23967.283,E2 -23967.283} C_VEL
LIN {X 0,Y 173.879,Z 461.21,A -85,B 0,C 180,E1 -23968.005,E2 -23968.005} C_VEL
LIN {X 0,Y 176.211,Z 457.698,A -85,B 0,C 180,E1 -23969.117,E2 -23969.117} C_VEL
LIN {X 0,Y 178.839,Z 451.74,A -85,B 0,C 180,E1 -23970.134,E2 -23970.134} C_VEL
LIN {X 0,Y 182.341,Z 441.238,A -85,B 0,C 180,E1 -23971.21,E2 -23971.21} C_VEL
LIN {X 0,Y 185.362,Z 430.748,A -85,B 0,C 180,E1 -23971.978,E2 -23971.978} C_VEL
LIN {X 0,Y 188.435,Z 426.154,A -85,B 0,C 180,E1 -23973.136,E2 -23973.136} C_VEL
LIN {X 0,Y 188.878,Z 425.347,A -85,B 0,C 180,E1 -23973.288,E2 -23973.288} C_VEL
LIN {X 0,Y 189.932,Z 425.666,A -85,B 0,C 180,E1 -23973.792,E2 -23973.792} C_VEL
LIN {X 0,Y 194.535,Z 433.636,A -85,B 0,C 180,E1 -23976.264,E2 -23976.264} C_VEL
LIN {X 0,Y 199.464,Z 444.82,A -85,B 0,C 180,E1 -23978.794,E2 -23978.794} C_VEL
LIN {X 0,Y 200.895,Z 448.486,A -85,B 0,C 180,E1 -23979.503,E2 -23979.503} C_VEL
LIN {X 0,Y 196.802,Z 503.422,A -85,B 0,C 180,E1 -23981.202,E2 -23981.202} C_VEL
LIN {X 0,Y 194.756,Z 517.355,A -85,B 0,C 180,E1 -23981.899,E2 -23981.899} C_VEL
LIN {X 0,Y 191.985,Z 530.878,A -85,B 0,C 180,E1 -23982.93,E2 -23982.93} C_VEL
LIN {X 0,Y 188.678,Z 543.167,A -85,B 0,C 180,E1 -23984.186,E2 -23984.186} C_VEL
LIN {X 0,Y 184.443,Z 556.045,A -85,B 0,C 180,E1 -23985.937,E2 -23985.937} C_VEL
LIN {X 0,Y 180.093,Z 567.597,A -85,B 0,C 180,E1 -23988.018,E2 -23988.018} C_VEL
LIN {X 0,Y 174.838,Z 579.4,A -85,B 0,C 180,E1 -23990.716,E2 -23990.716} C_VEL
LIN {X 0,Y 169.478,Z 589.827,A -85,B 0,C 180,E1 -23993.773,E2 -23993.773} C_VEL
LIN {X 0,Y 164.739,Z 598.424,A -85,B 0,C 180,E1 -23997.044,E2 -23997.044} C_VEL
LIN {X 0,Y 159.819,Z 606.662,A -85,B 0,C 180,E1 -24001.067,E2 -24001.067} C_VEL
LIN {X 0,Y 156.397,Z 612.407,A -85,B 0,C 180,E1 -24004.725,E2 -24004.725} C_VEL
LIN {X 0,Y 153.452,Z 617.125,A -85,B 0,C 180,E1 -24008.503,E2 -24008.503} C_VEL
LIN {X 0,Y 151.047,Z 620.949,A -85,B 0,C 180,E1 -24012.392,E2 -24012.392} C_VEL
LIN {X 0,Y 149.413,Z 623.884,A -85,B 0,C 180,E1 -24016.393,E2 -24016.393} C_VEL
LIN {X 0,Y 148.1,Z 626.58,A -85,B 0,C 180,E1 -24021.811,E2 -24021.811} C_VEL
LIN {X 0,Y 147.573,Z 627.928,A -85,B 0,C 180,E1 -24027.266,E2 -24027.266} C_VEL
LIN {X 0,Y 147.597,Z 628.082,A -85,B 0,C 180,E1 -24030.609,E2 -24030.609} C_VEL
LIN {X 0,Y 147.725,Z 627.473,A -85,B 0,C 180,E1 -24035.456,E2 -24035.456} C_VEL
LIN {X 0,Y 148.599,Z 625.506,A -85,B 0,C 180,E1 -24040.901,E2 -24040.901} C_VEL
LIN {X 0,Y 150.416,Z 622.155,A -85,B 0,C 180,E1 -24046.276,E2 -24046.276} C_VEL
LIN {X 0,Y 153.404,Z 617.315,A -85,B 0,C 180,E1 -24051.496,E2 -24051.496} C_VEL
LIN {X 0,Y 157.338,Z 610.845,A -85,B 0,C 180,E1 -24056.526,E2 -24056.526} C_VEL
LIN {X 0,Y 161.723,Z 603.639,A -85,B 0,C 180,E1 -24060.7,E2 -24060.7} C_VEL
LIN {X 0,Y 166.952,Z 594.718,A -85,B 0,C 180,E1 -24064.627,E2 -24064.627} C_VEL
LIN {X 0,Y 171.986,Z 585.346,A -85,B 0,C 180,E1 -24067.799,E2 -24067.799} C_VEL
LIN {X 0,Y 177.116,Z 574.964,A -85,B 0,C 180,E1 -24070.519,E2 -24070.519} C_VEL
LIN {X 0,Y 181.841,Z 563.516,A -85,B 0,C 180,E1 -24072.93,E2 -24072.93} C_VEL
LIN {X 0,Y 186.446,Z 550.811,A -85,B 0,C 180,E1 -24074.968,E2 -24074.968} C_VEL
LIN {X 0,Y 190.205,Z 538.433,A -85,B 0,C 180,E1 -24076.475,E2 -24076.475} C_VEL
LIN {X 0,Y 193.51,Z 524.698,A -85,B 0,C 180,E1 -24077.725,E2 -24077.725} C_VEL
LIN {X 0,Y 196.086,Z 510.361,A -85,B 0,C 180,E1 -24078.622,E2 -24078.622} C_VEL
LIN {X 0,Y 197.629,Z 496.092,A -85,B 0,C 180,E1 -24079.199,E2 -24079.199} C_VEL
LIN {X 0,Y 201.017,Z 449.507,A -85,B 0,C 180,E1 -24080.596,E2 -24080.596} C_VEL
LIN {X 0,Y 200.807,Z 447.959,A -85,B 0,C 180,E1 -24080.755,E2 -24080.755} C_VEL
LIN {X 0,Y 196.588,Z 438.005,A -85,B 0,C 180,E1 -24082.874,E2 -24082.874} C_VEL
LIN {X 0,Y 193.331,Z 431.276,A -85,B 0,C 180,E1 -24084.592,E2 -24084.592} C_VEL
LIN {X 0,Y 187.811,Z 422.151,A -85,B 0,C 180,E1 -24087.673,E2 -24087.673} C_VEL
LIN {X 0,Y 183.35,Z 415.411,A -85,B 0,C 180,E1 -24090.474,E2 -24090.474} C_VEL
LIN {X 0,Y 180.412,Z 411.188,A -85,B 0,C 180,E1 -24092.524,E2 -24092.524} C_VEL
LIN {X 0,Y 178.114,Z 407.97,A -85,B 0,C 180,E1 -24094.276,E2 -24094.276} C_VEL
LIN {X 0,Y 174.943,Z 403.641,A -85,B 0,C 180,E1 -24096.97,E2 -24096.97} C_VEL
LIN {X 0,Y 172.056,Z 400.21,A -85,B 0,C 180,E1 -24099.756,E2 -24099.756} C_VEL
LIN {X 0,Y 171.118,Z 398.691,A -85,B 0,C 180,E1 -24100.818,E2 -24100.818} C_VEL
LIN {X 0,Y 168.522,Z 396.068,A -85,B 0,C 180,E1 -24103.942,E2 -24103.942} C_VEL
LIN {X 0,Y 167.227,Z 393.469,A -85,B 0,C 180,E1 -24106.016,E2 -24106.016} C_VEL
LIN {X 0,Y 164.521,Z 391.395,A -85,B 0,C 180,E1 -24111.092,E2 -24111.092} C_VEL
LIN {X 0,Y 163.115,Z 388.187,A -85,B 0,C 180,E1 -24117.376,E2 -24117.376} C_VEL
LIN {X 0,Y 163.058,Z 387.594,A -85,B 0,C 180,E1 -24118.765,E2 -24118.765} C_VEL
LIN {X 0,Y 163.106,Z 387.645,A -85,B 0,C 180,E1 -24121.852,E2 -24121.852} C_VEL
LIN {X 0,Y 163.545,Z 389.856,A -85,B 0,C 180,E1 -24125.626,E2 -24125.626} C_VEL
LIN {X 0,Y 166.886,Z 393.334,A -85,B 0,C 180,E1 -24133.392,E2 -24133.392} C_VEL
LIN {X 0,Y 167.353,Z 393.809,A -85,B 0,C 180,E1 -24134.128,E2 -24134.128} C_VEL
LIN {X 0,Y 169.102,Z 396.88,A -85,B 0,C 180,E1 -24136.758,E2 -24136.758} C_VEL
LIN {X 0,Y 171.494,Z 399.194,A -85,B 0,C 180,E1 -24139.515,E2 -24139.515} C_VEL
LIN {X 0,Y 173.841,Z 402.614,A -85,B 0,C 180,E1 -24141.96,E2 -24141.96} C_VEL
LIN {X 0,Y 175.505,Z 404.422,A -85,B 0,C 180,E1 -24143.449,E2 -24143.449} C_VEL
LIN {X 0,Y 179.301,Z 409.597,A -85,B 0,C 180,E1 -24146.557,E2 -24146.557} C_VEL
LIN {X 0,Y 182.664,Z 414.438,A -85,B 0,C 180,E1 -24148.978,E2 -24148.978} C_VEL
LIN {X 0,Y 185.904,Z 419.218,A -85,B 0,C 180,E1 -24151.082,E2 -24151.082} C_VEL
LIN {X 0,Y 189.115,Z 424.485,A -85,B 0,C 180,E1 -24153.018,E2 -24153.018} C_VEL
LIN {X 0,Y 193.519,Z 433.309,A -85,B 0,C 180,E1 -24155.526,E2 -24155.526} C_VEL
LIN {X 0,Y 198.386,Z 444.261,A -85,B 0,C 180,E1 -24158.08,E2 -24158.08} C_VEL
LIN {X 0,Y 200.861,Z 450.684,A -85,B 0,C 180,E1 -24159.327,E2 -24159.327} C_VEL
LIN {X 0,Y 198.122,Z 490.379,A -85,B 0,C 180,E1 -24160.567,E2 -24160.567} C_VEL
LIN {X 0,Y 196.553,Z 508.017,A -85,B 0,C 180,E1 -24161.152,E2 -24161.152} C_VEL
LIN {X 0,Y 194.263,Z 522.578,A -85,B 0,C 180,E1 -24161.94,E2 -24161.94} C_VEL
LIN {X 0,Y 194.028,Z 523.774,A -85,B 0,C 180,E1 -24162.015,E2 -24162.015} C_VEL
LIN {X 0,Y 192.403,Z 529.402,A -85,B 0,C 180,E1 -24162.262,E2 -24162.262} C_VEL
LIN {X 0,Y 188.242,Z 538.399,A -85,B 0,C 180,E1 -24162.414,E2 -24162.414} C_VEL
LIN {X 0,Y 183.695,Z 547.128,A -85,B 0,C 180,E1 -24162.735,E2 -24162.735} C_VEL
LIN {X 0,Y 181.479,Z 552.331,A -85,B 0,C 180,E1 -24163.258,E2 -24163.258} C_VEL
LIN {X 0,Y 176.854,Z 564.521,A -85,B 0,C 180,E1 -24165.146,E2 -24165.146} C_VEL
LIN {X 0,Y 171.608,Z 576.616,A -85,B 0,C 180,E1 -24167.631,E2 -24167.631} C_VEL
LIN {X 0,Y 166.021,Z 587.744,A -85,B 0,C 180,E1 -24170.587,E2 -24170.587} C_VEL
LIN {X 0,Y 160.666,Z 597.162,A -85,B 0,C 180,E1 -24173.811,E2 -24173.811} C_VEL
LIN {X 0,Y 155.182,Z 606.134,A -85,B 0,C 180,E1 -24177.855,E2 -24177.855} C_VEL
LIN {X 0,Y 150.517,Z 613.385,A -85,B 0,C 180,E1 -24182.17,E2 -24182.17} C_VEL
LIN {X 0,Y 147.322,Z 618.469,A -85,B 0,C 180,E1 -24186.083,E2 -24186.083} C_VEL
LIN {X 0,Y 143.89,Z 623.717,A -85,B 0,C 180,E1 -24191.494,E2 -24191.494} C_VEL
LIN {X 0,Y 142.146,Z 626.661,A -85,B 0,C 180,E1 -24195.692,E2 -24195.692} C_VEL
LIN {X 0,Y 140.834,Z 629.349,A -85,B 0,C 180,E1 -24201.394,E2 -24201.394} C_VEL
LIN {X 0,Y 140.419,Z 630.674,A -85,B 0,C 180,E1 -24207.135,E2 -24207.135} C_VEL
LIN {X 0,Y 140.484,Z 630.835,A -85,B 0,C 180,E1 -24210.004,E2 -24210.004} C_VEL
LIN {X 0,Y 140.548,Z 630.151,A -85,B 0,C 180,E1 -24215.744,E2 -24215.744} C_VEL
LIN {X 0,Y 141.38,Z 628.123,A -85,B 0,C 180,E1 -24221.473,E2 -24221.473} C_VEL
LIN {X 0,Y 143.194,Z 624.706,A -85,B 0,C 180,E1 -24227.131,E2 -24227.131} C_VEL
LIN {X 0,Y 146.354,Z 619.802,A -85,B 0,C 180,E1 -24232.596,E2 -24232.596} C_VEL
LIN {X 0,Y 150.687,Z 613.256,A -85,B 0,C 180,E1 -24237.805,E2 -24237.805} C_VEL
LIN {X 0,Y 153.01,Z 610.067,A -85,B 0,C 180,E1 -24239.782,E2 -24239.782} C_VEL
LIN {X 0,Y 160.136,Z 610.474,A -85,B 0,C 180,E1 -24244.792,E2 -24244.792} C_VEL
LIN {X 0,Y 168.13,Z 609.751,A -85,B 0,C 180,E1 -24248.834,E2 -24248.834} C_VEL
LIN {X 0,Y 177.221,Z 607.95,A -85,B 0,C 180,E1 -24252.393,E2 -24252.393} C_VEL
LIN {X 0,Y 187.404,Z 605.023,A -85,B 0,C 180,E1 -24255.445,E2 -24255.445} C_VEL
LIN {X 0,Y 192.776,Z 603.123,A -85,B 0,C 180,E1 -24256.818,E2 -24256.818} C_VEL
LIN {X 0,Y 193.021,Z 602.945,A -85,B 0,C 180,E1 -24257.434,E2 -24257.434} C_VEL
LIN {X 0,Y 181.343,Z 605.668,A -85,B 0,C 180,E1 -24260.819,E2 -24260.819} C_VEL
LIN {X 0,Y 175.163,Z 606.445,A -85,B 0,C 180,E1 -24262.999,E2 -24262.999} C_VEL
LIN {X 0,Y 166.483,Z 606.606,A -85,B 0,C 180,E1 -24266.716,E2 -24266.716} C_VEL
LIN {X 0,Y 158.92,Z 605.478,A -85,B 0,C 180,E1 -24270.892,E2 -24270.892} C_VEL
LIN {X 0,Y 152.537,Z 603.055,A -85,B 0,C 180,E1 -24275.502,E2 -24275.502} C_VEL
LIN {X 0,Y 147.905,Z 599.385,A -85,B 0,C 180,E1 -24280.572,E2 -24280.572} C_VEL
LIN {X 0,Y 144.616,Z 594.345,A -85,B 0,C 180,E1 -24285.937,E2 -24285.937} C_VEL
LIN {X 0,Y 143.03,Z 589.168,A -85,B 0,C 180,E1 -24290.405,E2 -24290.405} C_VEL
LIN {X 0,Y 142.465,Z 582.74,A -85,B 0,C 180,E1 -24295.048,E2 -24295.048} C_VEL
LIN {X 0,Y 142.374,Z 575.484,A -85,B 0,C 180,E1 -24299.293,E2 -24299.293} C_VEL
LIN {X 0,Y 142.535,Z 568.228,A -85,B 0,C 180,E1 -24302.826,E2 -24302.826} C_VEL
LIN {X 0,Y 142.89,Z 559.458,A -85,B 0,C 180,E1 -24306.354,E2 -24306.354} C_VEL
LIN {X 0,Y 143.487,Z 549.254,A -85,B 0,C 180,E1 -24309.765,E2 -24309.765} C_VEL
LIN {X 0,Y 144.3,Z 538.165,A -85,B 0,C 180,E1 -24312.804,E2 -24312.804} C_VEL
LIN {X 0,Y 144.709,Z 532.514,A -85,B 0,C 180,E1 -24314.144,E2 -24314.144} C_VEL
LIN {X 0,Y 144.564,Z 533.324,A -85,B 0,C 180,E1 -24314.428,E2 -24314.428} C_VEL
LIN {X 0,Y 144.617,Z 533.763,A -85,B 0,C 180,E1 -24314.782,E2 -24314.782} C_VEL
LIN {X 0,Y 145.025,Z 533.876,A -85,B 0,C 180,E1 -24315.458,E2 -24315.458} C_VEL
LIN {X 0,Y 147.039,Z 531.799,A -85,B 0,C 180,E1 -24317.06,E2 -24317.06} C_VEL
LIN {X 0,Y 149.771,Z 527.628,A -85,B 0,C 180,E1 -24318.466,E2 -24318.466} C_VEL
LIN {X 0,Y 151.068,Z 525.318,A -85,B 0,C 180,E1 -24319.006,E2 -24319.006} C_VEL
LIN {X 0,Y 154.673,Z 521.662,A -85,B 0,C 180,E1 -24321.46,E2 -24321.46} C_VEL
LIN {X 0,Y 157.326,Z 517.507,A -85,B 0,C 180,E1 -24322.704,E2 -24322.704} C_VEL
LIN {X 0,Y 160.414,Z 511.024,A -85,B 0,C 180,E1 -24323.854,E2 -24323.854} C_VEL
LIN {X 0,Y 163.482,Z 502.205,A -85,B 0,C 180,E1 -24324.817,E2 -24324.817} C_VEL
LIN {X 0,Y 164.085,Z 500.283,A -85,B 0,C 180,E1 -24325.04,E2 -24325.04} C_VEL
LIN {X 0,Y 166.247,Z 496.826,A -85,B 0,C 180,E1 -24326.207,E2 -24326.207} C_VEL
LIN {X 0,Y 169.192,Z 489.8,A -85,B 0,C 180,E1 -24327.545,E2 -24327.545} C_VEL
LIN {X 0,Y 172.836,Z 478.315,A -85,B 0,C 180,E1 -24328.828,E2 -24328.828} C_VEL
LIN {X 0,Y 176.419,Z 465.437,A -85,B 0,C 180,E1 -24329.866,E2 -24329.866} C_VEL
LIN {X 0,Y 179.188,Z 460.758,A -85,B 0,C 180,E1 -24331.022,E2 -24331.022} C_VEL
LIN {X 0,Y 182.406,Z 453.262,A -85,B 0,C 180,E1 -24332.129,E2 -24332.129} C_VEL
LIN {X 0,Y 186.617,Z 440.346,A -85,B 0,C 180,E1 -24333.259,E2 -24333.259} C_VEL
LIN {X 0,Y 188.266,Z 434.86,A -85,B 0,C 180,E1 -24333.65,E2 -24333.65} C_VEL
LIN {X 0,Y 189.011,Z 434.701,A -85,B 0,C 180,E1 -24333.979,E2 -24333.979} C_VEL
LIN {X 0,Y 191.94,Z 440.444,A -85,B 0,C 180,E1 -24335.623,E2 -24335.623} C_VEL
LIN {X 0,Y 196.249,Z 450.759,A -85,B 0,C 180,E1 -24337.955,E2 -24337.955} C_VEL
LIN {X 0,Y 193.932,Z 482.133,A -85,B 0,C 180,E1 -24338.918,E2 -24338.918} C_VEL
LIN {X 0,Y 191.994,Z 504.939,A -85,B 0,C 180,E1 -24339.665,E2 -24339.665} C_VEL
LIN {X 0,Y 189.84,Z 518.955,A -85,B 0,C 180,E1 -24340.422,E2 -24340.422} C_VEL
LIN {X 0,Y 186.628,Z 533.21,A -85,B 0,C 180,E1 -24341.54,E2 -24341.54} C_VEL
LIN {X 0,Y 183.267,Z 545.003,A -85,B 0,C 180,E1 -24342.823,E2 -24342.823} C_VEL
LIN {X 0,Y 178.878,Z 557.541,A -85,B 0,C 180,E1 -24344.588,E2 -24344.588} C_VEL
LIN {X 0,Y 173.802,Z 570.148,A -85,B 0,C 180,E1 -24346.967,E2 -24346.967} C_VEL
LIN {X 0,Y 168.438,Z 581.385,A -85,B 0,C 180,E1 -24349.7,E2 -24349.7} C_VEL
LIN {X 0,Y 162.911,Z 591.432,A -85,B 0,C 180,E1 -24352.842,E2 -24352.842} C_VEL
LIN {X 0,Y 158.015,Z 599.772,A -85,B 0,C 180,E1 -24356.219,E2 -24356.219} C_VEL
LIN {X 0,Y 153.609,Z 606.732,A -85,B 0,C 180,E1 -24359.779,E2 -24359.779} C_VEL
LIN {X 0,Y 149.981,Z 612.476,A -85,B 0,C 180,E1 -24363.562,E2 -24363.562} C_VEL
LIN {X 0,Y 146.854,Z 617.194,A -85,B 0,C 180,E1 -24367.485,E2 -24367.485} C_VEL
LIN {X 0,Y 143.612,Z 622.076,A -85,B 0,C 180,E1 -24372.921,E2 -24372.921} C_VEL
LIN {X 0,Y 141.635,Z 625.472,A -85,B 0,C 180,E1 -24378.548,E2 -24378.548} C_VEL
LIN {X 0,Y 140.655,Z 627.488,A -85,B 0,C 180,E1 -24384.26,E2 -24384.26} C_VEL
LIN {X 0,Y 140.524,Z 628.172,A -85,B 0,C 180,E1 -24389.996,E2 -24389.996} C_VEL
LIN {X 0,Y 140.653,Z 627.54,A -85,B 0,C 180,E1 -24395.731,E2 -24395.731} C_VEL
LIN {X 0,Y 141.621,Z 625.573,A -85,B 0,C 180,E1 -24401.445,E2 -24401.445} C_VEL
LIN {X 0,Y 143.57,Z 622.221,A -85,B 0,C 180,E1 -24407.076,E2 -24407.076} C_VEL
LIN {X 0,Y 146.802,Z 617.381,A -85,B 0,C 180,E1 -24412.514,E2 -24412.514} C_VEL
LIN {X 0,Y 150.971,Z 610.912,A -85,B 0,C 180,E1 -24417.739,E2 -24417.739} C_VEL
LIN {X 0,Y 155.635,Z 603.705,A -85,B 0,C 180,E1 -24422.04,E2 -24422.04} C_VEL
LIN {X 0,Y 161.149,Z 594.783,A -85,B 0,C 180,E1 -24426.064,E2 -24426.064} C_VEL
LIN {X 0,Y 166.431,Z 585.411,A -85,B 0,C 180,E1 -24429.297,E2 -24429.297} C_VEL
LIN {X 0,Y 171.748,Z 575.076,A -85,B 0,C 180,E1 -24432.049,E2 -24432.049} C_VEL
LIN {X 0,Y 176.545,Z 563.962,A -85,B 0,C 180,E1 -24434.432,E2 -24434.432} C_VEL
LIN {X 0,Y 180.926,Z 552.454,A -85,B 0,C 180,E1 -24436.337,E2 -24436.337} C_VEL
LIN {X 0,Y 184.836,Z 540.481,A -85,B 0,C 180,E1 -24437.849,E2 -24437.849} C_VEL
LIN {X 0,Y 188.25,Z 527.356,A -85,B 0,C 180,E1 -24439.107,E2 -24439.107} C_VEL
LIN {X 0,Y 191.044,Z 513.159,A -85,B 0,C 180,E1 -24440.06,E2 -24440.06} C_VEL
LIN {X 0,Y 192.748,Z 499.866,A -85,B 0,C 180,E1 -24440.657,E2 -24440.657} C_VEL
LIN {X 0,Y 196.378,Z 451.997,A -85,B 0,C 180,E1 -24442.13,E2 -24442.13} C_VEL
LIN {X 0,Y 196.288,Z 450.647,A -85,B 0,C 180,E1 -24442.243,E2 -24442.243} C_VEL
LIN {X 0,Y 191.103,Z 438.352,A -85,B 0,C 180,E1 -24445.086,E2 -24445.086} C_VEL
LIN {X 0,Y 185.531,Z 428.663,A -85,B 0,C 180,E1 -24448.332,E2 -24448.332} C_VEL
LIN {X 0,Y 181.026,Z 421.587,A -85,B 0,C 180,E1 -24451.297,E2 -24451.297} C_VEL
LIN {X 0,Y 177.975,Z 417.103,A -85,B 0,C 180,E1 -24453.546,E2 -24453.546} C_VEL
LIN {X 0,Y 176.093,Z 414.344,A -85,B 0,C 180,E1 -24455.067,E2 -24455.067} C_VEL
LIN {X 0,Y 172.898,Z 409.951,A -85,B 0,C 180,E1 -24457.929,E2 -24457.929} C_VEL
LIN {X 0,Y 170.147,Z 406.312,A -85,B 0,C 180,E1 -24460.799,E2 -24460.799} C_VEL
LIN {X 0,Y 169.495,Z 405.355,A -85,B 0,C 180,E1 -24461.569,E2 -24461.569} C_VEL
LIN {X 0,Y 166.933,Z 402.418,A -85,B 0,C 180,E1 -24464.9,E2 -24464.9} C_VEL
LIN {X 0,Y 165.796,Z 400.287,A -85,B 0,C 180,E1 -24466.83,E2 -24466.83} C_VEL
LIN {X 0,Y 163.052,Z 397.688,A -85,B 0,C 180,E1 -24472.804,E2 -24472.804} C_VEL
LIN {X 0,Y 162.208,Z 395.014,A -85,B 0,C 180,E1 -24477.982,E2 -24477.982} C_VEL
LIN {X 0,Y 162.193,Z 394.643,A -85,B 0,C 180,E1 -24478.758,E2 -24478.758} C_VEL
LIN {X 0,Y 162.218,Z 394.763,A -85,B 0,C 180,E1 -24481.707,E2 -24481.707} C_VEL
LIN {X 0,Y 162.622,Z 396.886,A -85,B 0,C 180,E1 -24485.424,E2 -24485.424} C_VEL
LIN {X 0,Y 166.058,Z 400.695,A -85,B 0,C 180,E1 -24493.538,E2 -24493.538} C_VEL
LIN {X 0,Y 168.124,Z 404.113,A -85,B 0,C 180,E1 -24496.702,E2 -24496.702} C_VEL
LIN {X 0,Y 169.989,Z 406.02,A -85,B 0,C 180,E1 -24498.922,E2 -24498.922} C_VEL
LIN {X 0,Y 172.407,Z 409.477,A -85,B 0,C 180,E1 -24501.523,E2 -24501.523} C_VEL
LIN {X 0,Y 173.781,Z 411.106,A -85,B 0,C 180,E1 -24502.812,E2 -24502.812} C_VEL
LIN {X 0,Y 177.238,Z 415.994,A -85,B 0,C 180,E1 -24505.782,E2 -24505.782} C_VEL
LIN {X 0,Y 181.845,Z 422.742,A -85,B 0,C 180,E1 -24509.175,E2 -24509.175} C_VEL
LIN {X 0,Y 185.675,Z 429.055,A -85,B 0,C 180,E1 -24511.681,E2 -24511.681} C_VEL
LIN {X 0,Y 190.123,Z 438.263,A -85,B 0,C 180,E1 -24514.394,E2 -24514.394} C_VEL
LIN {X 0,Y 194.579,Z 448.669,A -85,B 0,C 180,E1 -24516.894,E2 -24516.894} C_VEL
LIN {X 0,Y 196.282,Z 453.198,A -85,B 0,C 180,E1 -24517.815,E2 -24517.815} C_VEL
LIN {X 0,Y 193.436,Z 491.89,A -85,B 0,C 180,E1 -24519.008,E2 -24519.008} C_VEL
LIN {X 0,Y 191.859,Z 508.906,A -85,B 0,C 180,E1 -24519.607,E2 -24519.607} C_VEL
LIN {X 0,Y 189.449,Z 523.282,A -85,B 0,C 180,E1 -24520.396,E2 -24520.396} C_VEL
LIN {X 0,Y 186.357,Z 536.467,A -85,B 0,C 180,E1 -24521.455,E2 -24521.455} C_VEL
LIN {X 0,Y 182.358,Z 549.85,A -85,B 0,C 180,E1 -24522.93,E2 -24522.93} C_VEL
LIN {X 0,Y 181.479,Z 552.331,A -85,B 0,C 180,E1 -24523.258,E2 -24523.258} C_VEL
LIN {X 0,Y 179.147,Z 557.525,A -85,B 0,C 180,E1 -24523.845,E2 -24523.845} C_VEL
LIN {X 0,Y 173.878,Z 565.65,A -85,B 0,C 180,E1 -24524.534,E2 -24524.534} C_VEL
LIN {X 0,Y 168.387,Z 573.447,A -85,B 0,C 180,E1 -24525.416,E2 -24525.416} C_VEL
LIN {X 0,Y 165.741,Z 577.952,A -85,B 0,C 180,E1 -24526.313,E2 -24526.313} C_VEL
LIN {X 0,Y 160.584,Z 587.679,A -85,B 0,C 180,E1 -24528.974,E2 -24528.974} C_VEL
LIN {X 0,Y 154.955,Z 597.097,A -85,B 0,C 180,E1 -24532.25,E2 -24532.25} C_VEL
LIN {X 0,Y 149.181,Z 606.068,A -85,B 0,C 180,E1 -24536.394,E2 -24536.394} C_VEL
LIN {X 0,Y 144.228,Z 613.318,A -85,B 0,C 180,E1 -24540.843,E2 -24540.843} C_VEL
LIN {X 0,Y 140.827,Z 618.403,A -85,B 0,C 180,E1 -24544.905,E2 -24544.905} C_VEL
LIN {X 0,Y 137.145,Z 623.65,A -85,B 0,C 180,E1 -24550.548,E2 -24550.548} C_VEL
LIN {X 0,Y 135.252,Z 626.594,A -85,B 0,C 180,E1 -24554.946,E2 -24554.946} C_VEL
LIN {X 0,Y 133.809,Z 629.282,A -85,B 0,C 180,E1 -24560.939,E2 -24560.939} C_VEL
LIN {X 0,Y 133.326,Z 630.607,A -85,B 0,C 180,E1 -24566.983,E2 -24566.983} C_VEL
LIN {X 0,Y 133.391,Z 630.768,A -85,B 0,C 180,E1 -24570.005,E2 -24570.005} C_VEL
LIN {X 0,Y 133.465,Z 630.083,A -85,B 0,C 180,E1 -24576.05,E2 -24576.05} C_VEL
LIN {X 0,Y 134.398,Z 628.055,A -85,B 0,C 180,E1 -24582.078,E2 -24582.078} C_VEL
LIN {X 0,Y 136.385,Z 624.638,A -85,B 0,C 180,E1 -24588.014,E2 -24588.014} C_VEL
LIN {X 0,Y 139.783,Z 619.734,A -85,B 0,C 180,E1 -24593.722,E2 -24593.722} C_VEL
LIN {X 0,Y 144.437,Z 613.187,A -85,B 0,C 180,E1 -24599.12,E2 -24599.12} C_VEL
LIN {X 0,Y 147.722,Z 609.109,A -85,B 0,C 180,E1 -24601.761,E2 -24601.761} C_VEL
LIN {X 0,Y 154.376,Z 609.833,A -85,B 0,C 180,E1 -24606.291,E2 -24606.291} C_VEL
LIN {X 0,Y 162.665,Z 609.589,A -85,B 0,C 180,E1 -24610.401,E2 -24610.401} C_VEL
LIN {X 0,Y 172.054,Z 608.302,A -85,B 0,C 180,E1 -24613.984,E2 -24613.984} C_VEL
LIN {X 0,Y 182.533,Z 605.931,A -85,B 0,C 180,E1 -24617.021,E2 -24617.021} C_VEL
LIN {X 0,Y 179.54,Z 606.347,A -85,B 0,C 180,E1 -24618.283,E2 -24618.283} C_VEL
LIN {X 0,Y 169.577,Z 607.229,A -85,B 0,C 180,E1 -24621.562,E2 -24621.562} C_VEL
LIN {X 0,Y 160.598,Z 606.859,A -85,B 0,C 180,E1 -24625.327,E2 -24625.327} C_VEL
LIN {X 0,Y 152.778,Z 605.254,A -85,B 0,C 180,E1 -24629.601,E2 -24629.601} C_VEL
LIN {X 0,Y 146.159,Z 602.379,A -85,B 0,C 180,E1 -24634.357,E2 -24634.357} C_VEL
LIN {X 0,Y 141.333,Z 598.264,A -85,B 0,C 180,E1 -24639.63,E2 -24639.63} C_VEL
LIN {X 0,Y 137.909,Z 592.767,A -85,B 0,C 180,E1 -24645.238,E2 -24645.238} C_VEL
LIN {X 0,Y 136.283,Z 587.075,A -85,B 0,C 180,E1 -24650.045,E2 -24650.045} C_VEL
LIN {X 0,Y 135.723,Z 580.392,A -85,B 0,C 180,E1 -24654.801,E2 -24654.801} C_VEL
LIN {X 0,Y 135.659,Z 572.748,A -85,B 0,C 180,E1 -24659.258,E2 -24659.258} C_VEL
LIN {X 0,Y 135.82,Z 564.973,A -85,B 0,C 180,E1 -24662.966,E2 -24662.966} C_VEL
LIN {X 0,Y 136.277,Z 554.641,A -85,B 0,C 180,E1 -24667.036,E2 -24667.036} C_VEL
LIN {X 0,Y 136.776,Z 545.513,A -85,B 0,C 180,E1 -24670.041,E2 -24670.041} C_VEL
LIN {X 0,Y 136.63,Z 545.948,A -85,B 0,C 180,E1 -24670.22,E2 -24670.22} C_VEL
LIN {X 0,Y 137.126,Z 546.409,A -85,B 0,C 180,E1 -24671.83,E2 -24671.83} C_VEL
LIN {X 0,Y 138.051,Z 545.599,A -85,B 0,C 180,E1 -24672.831,E2 -24672.831} C_VEL
LIN {X 0,Y 140.446,Z 542.781,A -85,B 0,C 180,E1 -24674.49,E2 -24674.49} C_VEL
LIN {X 0,Y 141.552,Z 541.253,A -85,B 0,C 180,E1 -24675.11,E2 -24675.11} C_VEL
LIN {X 0,Y 142.377,Z 540.396,A -85,B 0,C 180,E1 -24675.753,E2 -24675.753} C_VEL
LIN {X 0,Y 143.701,Z 539.578,A -85,B 0,C 180,E1 -24677.064,E2 -24677.064} C_VEL
LIN {X 0,Y 146.235,Z 537.188,A -85,B 0,C 180,E1 -24678.83,E2 -24678.83} C_VEL
LIN {X 0,Y 148.794,Z 533.846,A -85,B 0,C 180,E1 -24680.091,E2 -24680.091} C_VEL
LIN {X 0,Y 151.129,Z 530.472,A -85,B 0,C 180,E1 -24681.055,E2 -24681.055} C_VEL
LIN {X 0,Y 154.018,Z 527.774,A -85,B 0,C 180,E1 -24682.822,E2 -24682.822} C_VEL
LIN {X 0,Y 156.26,Z 524.999,A -85,B 0,C 180,E1 -24683.878,E2 -24683.878} C_VEL
LIN {X 0,Y 159.353,Z 520.163,A -85,B 0,C 180,E1 -24685.064,E2 -24685.064} C_VEL
LIN {X 0,Y 162.636,Z 513.561,A -85,B 0,C 180,E1 -24686.073,E2 -24686.073} C_VEL
LIN {X 0,Y 165.718,Z 505.5,A -85,B 0,C 180,E1 -24686.895,E2 -24686.895} C_VEL
LIN {X 0,Y 166.185,Z 504.503,A -85,B 0,C 180,E1 -24687.067,E2 -24687.067} C_VEL
LIN {X 0,Y 168.894,Z 499.822,A -85,B 0,C 180,E1 -24688.296,E2 -24688.296} C_VEL
LIN {X 0,Y 171.85,Z 493.02,A -85,B 0,C 180,E1 -24689.474,E2 -24689.474} C_VEL
LIN {X 0,Y 175.659,Z 481.469,A -85,B 0,C 180,E1 -24690.714,E2 -24690.714} C_VEL
LIN {X 0,Y 179.076,Z 469.515,A -85,B 0,C 180,E1 -24691.627,E2 -24691.627} C_VEL
LIN {X 0,Y 182.129,Z 464.224,A -85,B 0,C 180,E1 -24692.782,E2 -24692.782} C_VEL
LIN {X 0,Y 185.513,Z 456.461,A -85,B 0,C 180,E1 -24693.85,E2 -24693.85} C_VEL
LIN {X 0,Y 188.56,Z 447.634,A -85,B 0,C 180,E1 -24694.635,E2 -24694.635} C_VEL
LIN {X 0,Y 189.655,Z 448.026,A -85,B 0,C 180,E1 -24695.138,E2 -24695.138} C_VEL
LIN {X 0,Y 191.775,Z 453.385,A -85,B 0,C 180,E1 -24696.364,E2 -24696.364} C_VEL
LIN {X 0,Y 189.575,Z 481.957,A -85,B 0,C 180,E1 -24697.241,E2 -24697.241} C_VEL
LIN {X 0,Y 187.635,Z 504.403,A -85,B 0,C 180,E1 -24697.972,E2 -24697.972} C_VEL
LIN {X 0,Y 185.443,Z 518.27,A -85,B 0,C 180,E1 -24698.692,E2 -24698.692} C_VEL
LIN {X 0,Y 182.313,Z 532.156,A -85,B 0,C 180,E1 -24699.77,E2 -24699.77} C_VEL
LIN {X 0,Y 178.507,Z 545.076,A -85,B 0,C 180,E1 -24701.147,E2 -24701.147} C_VEL
LIN {X 0,Y 173.958,Z 557.613,A -85,B 0,C 180,E1 -24702.92,E2 -24702.92} C_VEL
LIN {X 0,Y 169.188,Z 569.047,A -85,B 0,C 180,E1 -24705.071,E2 -24705.071} C_VEL
LIN {X 0,Y 164.08,Z 579.541,A -85,B 0,C 180,E1 -24707.571,E2 -24707.571} C_VEL
LIN {X 0,Y 158.196,Z 589.967,A -85,B 0,C 180,E1 -24710.719,E2 -24710.719} C_VEL
LIN {X 0,Y 152.964,Z 598.564,A -85,B 0,C 180,E1 -24714.136,E2 -24714.136} C_VEL
LIN {X 0,Y 147.485,Z 606.801,A -85,B 0,C 180,E1 -24718.383,E2 -24718.383} C_VEL
LIN {X 0,Y 143.63,Z 612.545,A -85,B 0,C 180,E1 -24722.295,E2 -24722.295} C_VEL
LIN {X 0,Y 140.308,Z 617.262,A -85,B 0,C 180,E1 -24726.372,E2 -24726.372} C_VEL
LIN {X 0,Y 136.795,Z 622.145,A -85,B 0,C 180,E1 -24732.041,E2 -24732.041} C_VEL
LIN {X 0,Y 134.652,Z 625.541,A -85,B 0,C 180,E1 -24737.945,E2 -24737.945} C_VEL
LIN {X 0,Y 133.582,Z 627.555,A -85,B 0,C 180,E1 -24743.955,E2 -24743.955} C_VEL
LIN {X 0,Y 133.449,Z 628.239,A -85,B 0,C 180,E1 -24749.995,E2 -24749.995} C_VEL
LIN {X 0,Y 133.579,Z 627.607,A -85,B 0,C 180,E1 -24756.036,E2 -24756.036} C_VEL
LIN {X 0,Y 134.036,Z 626.792,A -85,B 0,C 180,E1 -24759.046,E2 -24759.046} C_VEL
LIN {X 0,Y 135.561,Z 624.142,A -85,B 0,C 180,E1 -24765.019,E2 -24765.019} C_VEL
LIN {X 0,Y 138.323,Z 620.062,A -85,B 0,C 180,E1 -24770.829,E2 -24770.829} C_VEL
LIN {X 0,Y 141.271,Z 616.024,A -85,B 0,C 180,E1 -24775.01,E2 -24775.01} C_VEL
LIN {X 0,Y 144.679,Z 610.978,A -85,B 0,C 180,E1 -24779.057,E2 -24779.057} C_VEL
LIN {X 0,Y 149.653,Z 603.77,A -85,B 0,C 180,E1 -24783.486,E2 -24783.486} C_VEL
LIN {X 0,Y 155.457,Z 594.848,A -85,B 0,C 180,E1 -24787.607,E2 -24787.607} C_VEL
LIN {X 0,Y 161.001,Z 585.475,A -85,B 0,C 180,E1 -24790.897,E2 -24790.897} C_VEL
LIN {X 0,Y 166.905,Z 574.345,A -85,B 0,C 180,E1 -24793.878,E2 -24793.878} C_VEL
LIN {X 0,Y 171.693,Z 563.642,A -85,B 0,C 180,E1 -24796.168,E2 -24796.168} C_VEL
LIN {X 0,Y 176.667,Z 550.935,A -85,B 0,C 180,E1 -24798.23,E2 -24798.23} C_VEL
LIN {X 0,Y 180.715,Z 538.555,A -85,B 0,C 180,E1 -24799.742,E2 -24799.742} C_VEL
LIN {X 0,Y 184.271,Z 524.815,A -85,B 0,C 180,E1 -24800.989,E2 -24800.989} C_VEL
LIN {X 0,Y 187.024,Z 510.472,A -85,B 0,C 180,E1 -24801.88,E2 -24801.88} C_VEL
LIN {X 0,Y 188.643,Z 496.529,A -85,B 0,C 180,E1 -24802.448,E2 -24802.448} C_VEL
LIN {X 0,Y 191.98,Z 453.644,A -85,B 0,C 180,E1 -24803.752,E2 -24803.752} C_VEL
LIN {X 0,Y 187.372,Z 442.627,A -85,B 0,C 180,E1 -24806.467,E2 -24806.467} C_VEL
LIN {X 0,Y 182.444,Z 433.803,A -85,B 0,C 180,E1 -24809.549,E2 -24809.549} C_VEL
LIN {X 0,Y 178.275,Z 427.091,A -85,B 0,C 180,E1 -24812.485,E2 -24812.485} C_VEL
LIN {X 0,Y 174.322,Z 420.945,A -85,B 0,C 180,E1 -24815.696,E2 -24815.696} C_VEL
LIN {X 0,Y 171.049,Z 416.368,A -85,B 0,C 180,E1 -24818.771,E2 -24818.771} C_VEL
LIN {X 0,Y 168.323,Z 412.462,A -85,B 0,C 180,E1 -24821.829,E2 -24821.829} C_VEL
LIN {X 0,Y 165.312,Z 408.649,A -85,B 0,C 180,E1 -24826.007,E2 -24826.007} C_VEL
LIN {X 0,Y 164.581,Z 407.171,A -85,B 0,C 180,E1 -24827.358,E2 -24827.358} C_VEL
LIN {X 0,Y 161.351,Z 402.742,A -85,B 0,C 180,E1 -24837.191,E2 -24837.191} C_VEL
LIN {X 0,Y 161.324,Z 401.722,A -85,B 0,C 180,E1 -24838.752,E2 -24838.752} C_VEL
LIN {X 0,Y 161.326,Z 401.833,A -85,B 0,C 180,E1 -24841.404,E2 -24841.404} C_VEL
LIN {X 0,Y 162.092,Z 404.712,A -85,B 0,C 180,E1 -24846.848,E2 -24846.848} C_VEL
LIN {X 0,Y 164.785,Z 407.547,A -85,B 0,C 180,E1 -24852.939,E2 -24852.939} C_VEL
LIN {X 0,Y 167.184,Z 411.344,A -85,B 0,C 180,E1 -24856.686,E2 -24856.686} C_VEL
LIN {X 0,Y 168.437,Z 412.725,A -85,B 0,C 180,E1 -24858.236,E2 -24858.236} C_VEL
LIN {X 0,Y 171.269,Z 416.617,A -85,B 0,C 180,E1 -24861.357,E2 -24861.357} C_VEL
LIN {X 0,Y 175.131,Z 422.244,A -85,B 0,C 180,E1 -24864.921,E2 -24864.921} C_VEL
LIN {X 0,Y 179.345,Z 428.647,A -85,B 0,C 180,E1 -24868.207,E2 -24868.207} C_VEL
LIN {X 0,Y 182.912,Z 434.763,A -85,B 0,C 180,E1 -24870.684,E2 -24870.684} C_VEL
LIN {X 0,Y 186.944,Z 443.493,A -85,B 0,C 180,E1 -24873.306,E2 -24873.306} C_VEL
LIN {X 0,Y 190.895,Z 453.18,A -85,B 0,C 180,E1 -24875.683,E2 -24875.683} C_VEL
LIN {X 0,Y 191.853,Z 455.772,A -85,B 0,C 180,E1 -24876.24,E2 -24876.24} C_VEL
LIN {X 0,Y 187.889,Z 504.82,A -85,B 0,C 180,E1 -24877.743,E2 -24877.743} C_VEL
LIN {X 0,Y 185.723,Z 519.415,A -85,B 0,C 180,E1 -24878.485,E2 -24878.485} C_VEL
LIN {X 0,Y 182.625,Z 533.016,A -85,B 0,C 180,E1 -24879.466,E2 -24879.466} C_VEL
LIN {X 0,Y 178.772,Z 546.253,A -85,B 0,C 180,E1 -24880.826,E2 -24880.826} C_VEL
LIN {X 0,Y 174.138,Z 559.013,A -85,B 0,C 180,E1 -24882.568,E2 -24882.568} C_VEL
LIN {X 0,Y 169.197,Z 570.615,A -85,B 0,C 180,E1 -24884.663,E2 -24884.663} C_VEL
LIN {X 0,Y 165.741,Z 577.952,A -85,B 0,C 180,E1 -24886.313,E2 -24886.313} C_VEL
LIN {X 0,Y 163.013,Z 582.372,A -85,B 0,C 180,E1 -24887.294,E2 -24887.294} C_VEL
LIN {X 0,Y 156.987,Z 589.279,A -85,B 0,C 180,E1 -24888.652,E2 -24888.652} C_VEL
LIN {X 0,Y 150.765,Z 595.745,A -85,B 0,C 180,E1 -24890.245,E2 -24890.245} C_VEL
LIN {X 0,Y 147.8,Z 599.416,A -85,B 0,C 180,E1 -24891.603,E2 -24891.603} C_VEL
LIN {X 0,Y 142.485,Z 607.12,A -85,B 0,C 180,E1 -24895.448,E2 -24895.448} C_VEL
LIN {X 0,Y 138.035,Z 613.252,A -85,B 0,C 180,E1 -24899.398,E2 -24899.398} C_VEL
LIN {X 0,Y 134.391,Z 618.336,A -85,B 0,C 180,E1 -24903.613,E2 -24903.613} C_VEL
LIN {X 0,Y 130.446,Z 623.584,A -85,B 0,C 180,E1 -24909.506,E2 -24909.506} C_VEL
LIN {X 0,Y 128.37,Z 626.527,A -85,B 0,C 180,E1 -24914.118,E2 -24914.118} C_VEL
LIN {X 0,Y 126.777,Z 629.215,A -85,B 0,C 180,E1 -24920.432,E2 -24920.432} C_VEL
LIN {X 0,Y 126.241,Z 630.54,A -85,B 0,C 180,E1 -24926.813,E2 -24926.813} C_VEL
LIN {X 0,Y 126.307,Z 630.701,A -85,B 0,C 180,E1 -24930.005,E2 -24930.005} C_VEL
LIN {X 0,Y 126.408,Z 630.016,A -85,B 0,C 180,E1 -24936.389,E2 -24936.389} C_VEL
LIN {X 0,Y 127.428,Z 627.986,A -85,B 0,C 180,E1 -24942.75,E2 -24942.75} C_VEL
LIN {X 0,Y 129.619,Z 624.569,A -85,B 0,C 180,E1 -24948.99,E2 -24948.99} C_VEL
LIN {X 0,Y 133.278,Z 619.665,A -85,B 0,C 180,E1 -24954.956,E2 -24954.956} C_VEL
LIN {X 0,Y 137.392,Z 614.205,A -85,B 0,C 180,E1 -24959.753,E2 -24959.753} C_VEL
LIN {X 0,Y 142.533,Z 608.039,A -85,B 0,C 180,E1 -24963.802,E2 -24963.802} C_VEL
LIN {X 0,Y 148.764,Z 608.989,A -85,B 0,C 180,E1 -24967.895,E2 -24967.895} C_VEL
LIN {X 0,Y 157.334,Z 609.205,A -85,B 0,C 180,E1 -24972.075,E2 -24972.075} C_VEL
LIN {X 0,Y 167.031,Z 608.425,A -85,B 0,C 180,E1 -24975.672,E2 -24975.672} C_VEL
LIN {X 0,Y 172.289,Z 607.647,A -85,B 0,C 180,E1 -24977.249,E2 -24977.249} C_VEL
LIN {X 0,Y 164.089,Z 607.796,A -85,B 0,C 180,E1 -24980.025,E2 -24980.025} C_VEL
LIN {X 0,Y 154.823,Z 606.903,A -85,B 0,C 180,E1 -24983.835,E2 -24983.835} C_VEL
LIN {X 0,Y 146.725,Z 604.809,A -85,B 0,C 180,E1 -24988.205,E2 -24988.205} C_VEL
LIN {X 0,Y 139.845,Z 601.488,A -85,B 0,C 180,E1 -24993.109,E2 -24993.109} C_VEL
LIN {X 0,Y 134.828,Z 596.934,A -85,B 0,C 180,E1 -24998.6,E2 -24998.6} C_VEL
LIN {X 0,Y 131.212,Z 590.813,A -85,B 0,C 180,E1 -25004.621,E2 -25004.621} C_VEL
LIN {X 0,Y 129.408,Z 583.487,A -85,B 0,C 180,E1 -25010.623,E2 -25010.623} C_VEL
LIN {X 0,Y 129.035,Z 576.606,A -85,B 0,C 180,E1 -25015.314,E2 -25015.314} C_VEL
LIN {X 0,Y 129.035,Z 568.138,A -85,B 0,C 180,E1 -25020,E2 -25020} C_VEL
LIN {X 0,Y 129.233,Z 559.589,A -85,B 0,C 180,E1 -25023.898,E2 -25023.898} C_VEL
LIN {X 0,Y 129.339,Z 556.436,A -85,B 0,C 180,E1 -25025.164,E2 -25025.164} C_VEL
LIN {X 0,Y 129.036,Z 557.246,A -85,B 0,C 180,E1 -25026.254,E2 -25026.254} C_VEL
LIN {X 0,Y 130.975,Z 555.556,A -85,B 0,C 180,E1 -25029.264,E2 -25029.264} C_VEL
LIN {X 0,Y 132.74,Z 553.485,A -85,B 0,C 180,E1 -25030.679,E2 -25030.679} C_VEL
LIN {X 0,Y 135.014,Z 551.944,A -85,B 0,C 180,E1 -25033.547,E2 -25033.547} C_VEL
LIN {X 0,Y 136.624,Z 550.522,A -85,B 0,C 180,E1 -25034.904,E2 -25034.904} C_VEL
LIN {X 0,Y 140.713,Z 546.198,A -85,B 0,C 180,E1 -25037.438,E2 -25037.438} C_VEL
LIN {X 0,Y 142.269,Z 545.179,A -85,B 0,C 180,E1 -25038.729,E2 -25038.729} C_VEL
LIN {X 0,Y 145.287,Z 542.575,A -85,B 0,C 180,E1 -25040.598,E2 -25040.598} C_VEL
LIN {X 0,Y 148.865,Z 538.383,A -85,B 0,C 180,E1 -25042.191,E2 -25042.191} C_VEL
LIN {X 0,Y 150.302,Z 536.487,A -85,B 0,C 180,E1 -25042.691,E2 -25042.691} C_VEL
LIN {X 0,Y 153.447,Z 533.553,A -85,B 0,C 180,E1 -25044.344,E2 -25044.344} C_VEL
LIN {X 0,Y 156.852,Z 529.79,A -85,B 0,C 180,E1 -25045.779,E2 -25045.779} C_VEL
LIN {X 0,Y 160.089,Z 525.227,A -85,B 0,C 180,E1 -25046.894,E2 -25046.894} C_VEL
LIN {X 0,Y 164.165,Z 518.021,A -85,B 0,C 180,E1 -25048.01,E2 -25048.01} C_VEL
LIN {X 0,Y 168.273,Z 508.607,A -85,B 0,C 180,E1 -25048.996,E2 -25048.996} C_VEL
LIN {X 0,Y 171.344,Z 503.546,A -85,B 0,C 180,E1 -25050.163,E2 -25050.163} C_VEL
LIN {X 0,Y 174.742,Z 496.114,A -85,B 0,C 180,E1 -25051.358,E2 -25051.358} C_VEL
LIN {X 0,Y 178.849,Z 484.048,A -85,B 0,C 180,E1 -25052.588,E2 -25052.588} C_VEL
LIN {X 0,Y 182.083,Z 473.23,A -85,B 0,C 180,E1 -25053.399,E2 -25053.399} C_VEL
LIN {X 0,Y 185.5,Z 467.12,A -85,B 0,C 180,E1 -25054.565,E2 -25054.565} C_VEL
LIN {X 0,Y 186.881,Z 464.118,A -85,B 0,C 180,E1 -25054.98,E2 -25054.98} C_VEL
LIN {X 0,Y 183.474,Z 503.689,A -85,B 0,C 180,E1 -25056.194,E2 -25056.194} C_VEL
LIN {X 0,Y 181.089,Z 518.348,A -85,B 0,C 180,E1 -25056.938,E2 -25056.938} C_VEL
LIN {X 0,Y 177.86,Z 532.231,A -85,B 0,C 180,E1 -25058.014,E2 -25058.014} C_VEL
LIN {X 0,Y 173.922,Z 545.149,A -85,B 0,C 180,E1 -25059.387,E2 -25059.387} C_VEL
LIN {X 0,Y 169.213,Z 557.685,A -85,B 0,C 180,E1 -25061.162,E2 -25061.162} C_VEL
LIN {X 0,Y 163.842,Z 569.95,A -85,B 0,C 180,E1 -25063.492,E2 -25063.492} C_VEL
LIN {X 0,Y 158.9,Z 579.612,A -85,B 0,C 180,E1 -25065.84,E2 -25065.84} C_VEL
LIN {X 0,Y 152.753,Z 590.037,A -85,B 0,C 180,E1 -25069.028,E2 -25069.028} C_VEL
LIN {X 0,Y 147.244,Z 598.634,A -85,B 0,C 180,E1 -25072.51,E2 -25072.51} C_VEL
LIN {X 0,Y 141.463,Z 606.87,A -85,B 0,C 180,E1 -25076.869,E2 -25076.869} C_VEL
LIN {X 0,Y 137.354,Z 612.614,A -85,B 0,C 180,E1 -25080.912,E2 -25080.912} C_VEL
LIN {X 0,Y 133.817,Z 617.331,A -85,B 0,C 180,E1 -25085.151,E2 -25085.151} C_VEL
LIN {X 0,Y 130.019,Z 622.214,A -85,B 0,C 180,E1 -25091.071,E2 -25091.071} C_VEL
LIN {X 0,Y 127.692,Z 625.609,A -85,B 0,C 180,E1 -25097.277,E2 -25097.277} C_VEL
LIN {X 0,Y 126.533,Z 627.623,A -85,B 0,C 180,E1 -25103.617,E2 -25103.617} C_VEL
LIN {X 0,Y 126.36,Z 628.306,A -85,B 0,C 180,E1 -25109.995,E2 -25109.995} C_VEL
LIN {X 0,Y 126.53,Z 627.674,A -85,B 0,C 180,E1 -25116.373,E2 -25116.373} C_VEL
LIN {X 0,Y 127.676,Z 625.707,A -85,B 0,C 180,E1 -25122.715,E2 -25122.715} C_VEL
LIN {X 0,Y 129.983,Z 622.355,A -85,B 0,C 180,E1 -25128.925,E2 -25128.925} C_VEL
LIN {X 0,Y 133.741,Z 617.514,A -85,B 0,C 180,E1 -25134.854,E2 -25134.854} C_VEL
LIN {X 0,Y 138.091,Z 611.571,A -85,B 0,C 180,E1 -25140.094,E2 -25140.094} C_VEL
LIN {X 0,Y 142.94,Z 604.95,A -85,B 0,C 180,E1 -25144.426,E2 -25144.426} C_VEL
LIN {X 0,Y 148.947,Z 596.279,A -85,B 0,C 180,E1 -25148.691,E2 -25148.691} C_VEL
LIN {X 0,Y 154.667,Z 587.205,A -85,B 0,C 180,E1 -25152.079,E2 -25152.079} C_VEL
LIN {X 0,Y 160.786,Z 576.482,A -85,B 0,C 180,E1 -25155.13,E2 -25155.13} C_VEL
LIN {X 0,Y 166.292,Z 564.996,A -85,B 0,C 180,E1 -25157.69,E2 -25157.69} C_VEL
LIN {X 0,Y 171.435,Z 552.578,A -85,B 0,C 180,E1 -25159.77,E2 -25159.77} C_VEL
LIN {X 0,Y 175.619,Z 540.602,A -85,B 0,C 180,E1 -25161.287,E2 -25161.287} C_VEL
LIN {X 0,Y 179.288,Z 527.473,A -85,B 0,C 180,E1 -25162.535,E2 -25162.535} C_VEL
LIN {X 0,Y 182.262,Z 513.27,A -85,B 0,C 180,E1 -25163.481,E2 -25163.481} C_VEL
LIN {X 0,Y 184.147,Z 499.262,A -85,B 0,C 180,E1 -25164.1,E2 -25164.1} C_VEL
LIN {X 0,Y 187.664,Z 456.305,A -85,B 0,C 180,E1 -25165.417,E2 -25165.417} C_VEL
LIN {X 0,Y 183.992,Z 447.341,A -85,B 0,C 180,E1 -25167.753,E2 -25167.753} C_VEL
LIN {X 0,Y 178.566,Z 437.387,A -85,B 0,C 180,E1 -25171.444,E2 -25171.444} C_VEL
LIN {X 0,Y 174.071,Z 430.021,A -85,B 0,C 180,E1 -25174.996,E2 -25174.996} C_VEL
LIN {X 0,Y 171.587,Z 426.299,A -85,B 0,C 180,E1 -25177.234,E2 -25177.234} C_VEL
LIN {X 0,Y 169.228,Z 422.745,A -85,B 0,C 180,E1 -25179.646,E2 -25179.646} C_VEL
LIN {X 0,Y 166.35,Z 418.618,A -85,B 0,C 180,E1 -25183.113,E2 -25183.113} C_VEL
LIN {X 0,Y 163.834,Z 415.038,A -85,B 0,C 180,E1 -25186.985,E2 -25186.985} C_VEL
LIN {X 0,Y 163.291,Z 414.037,A -85,B 0,C 180,E1 -25188.046,E2 -25188.046} C_VEL
LIN {X 0,Y 160.43,Z 409.174,A -85,B 0,C 180,E1 -25198.431,E2 -25198.431} C_VEL
LIN {X 0,Y 160.437,Z 408.721,A -85,B 0,C 180,E1 -25199.372,E2 -25199.372} C_VEL
LIN {X 0,Y 160.435,Z 408.932,A -85,B 0,C 180,E1 -25201.098,E2 -25201.098} C_VEL
LIN {X 0,Y 162.93,Z 413.784,A -85,B 0,C 180,E1 -25211.192,E2 -25211.192} C_VEL
LIN {X 0,Y 163.571,Z 414.454,A -85,B 0,C 180,E1 -25212.405,E2 -25212.405} C_VEL
LIN {X 0,Y 165.931,Z 418.224,A -85,B 0,C 180,E1 -25216.256,E2 -25216.256} C_VEL
LIN {X 0,Y 166.97,Z 419.491,A -85,B 0,C 180,E1 -25217.61,E2 -25217.61} C_VEL
LIN {X 0,Y 170.374,Z 424.444,A -85,B 0,C 180,E1 -25221.475,E2 -25221.475} C_VEL
LIN {X 0,Y 173.064,Z 428.504,A -85,B 0,C 180,E1 -25224.039,E2 -25224.039} C_VEL
LIN {X 0,Y 177.125,Z 434.955,A -85,B 0,C 180,E1 -25227.388,E2 -25227.388} C_VEL
